DATA_BLOCK "DB3323"
TITLE =STAZIONE ++ZNE05
{ S7_language := '22(1) Portoghese (Brasile)  01.09.2016  10:42:20' }
VERSION : 0.1


  STRUCT
   CM_ID : STRING  [8 ] := '=DCK_2';	//COMPOSITE MACHINE
   STATION_ID : STRING  [8 ] := '++ZNE05';	//STATION - TRATTO - ZONE
   ELEMENT_ID : STRING  [8 ];	//ELEMENT
   DB_ID : INT  := 3;	//DB SIZE or TYPE
   PART_STYLE : STRING  [12 ];	//PART STYLE ON LAST STATION
   ACT_CYCLE_TIME : INT ;	//ACTUAL CYCLE TIME FOR THIS STYLE
   COUNT_GOOD : INT ;	//COUNTER GOOD PIECES
   COUNT_SCRAP : INT ;	//COUNTER SCRAP PIECES
   SPARE_00 : ARRAY  [0 .. 15 ] OF //SPARE INTEGER
   INT ;
   SPARE_01 : ARRAY  [0 .. 17 ] OF //SPARE INTEGER
   INT ;
   CODE_EVENT : ARRAY  [0 .. 7 ] OF INT ;
EVENTS : STRUCT
   E0000 : BOOL ;	//=DCK_2++ZNE05+PTZ01-SB_09;EMERGÊNCIA ATIVADA - NO PTZ01;2
   E0001 : BOOL ;	//=DCK_2++ZNE05+PTZ02-SB_09;EMERGÊNCIA ATIVADA - NO PTZ02;2
   E0002 : BOOL ;	//=DCK_2++ZNE05;EMERGÊNCIA NÃO RESTAURADA EM ++ZNE05;2
   E0003 : BOOL ;	//=DCK_2++ZNE05;ÁREAS DE AJUSTE DE EMERGÊNCIA ++ZNE05 (++ZNE04/6/7);2
   E0004 : BOOL ;	//=DCK_2++ZNE05+HCZ01-KM_06;FALHA DO CONTATO DO FREIO TR_01;1
   E0005 : BOOL ;	//=DCK_2++ZNE05+HCZ01-KM_08;FALHA NO CONTATO DO FREIO TR_02;1
   E0006 : BOOL ;	//=DCK_2++ZNE05+HCZ01-DMC01;ANOMALIA DO MÓDULO SEGURO ET200S-FDI-FDO;2
   E0007 : BOOL ;	//=DCK_2++ZNE05+HKM01-DMC01;ANOMALIA DO MÓDULO SEGURO ET200S-FDI;2
   E0008 : BOOL ;	//=DCK_2++ZNE05+PTZ01-DMC01;ANOMALIA DO MÓDULO SEGURO ET200S-FDI;2
   E0009 : BOOL ;	//=DCK_2++ZNE05+PTZ02-DMC01;ANOMALIA DO MÓDULO SEGURO ET200S-FDI;2
   E0010 : BOOL ;	//=DCK_2++ZNE05+HKM02-DMC01;ANOMALIA DO MÓDULO SEGURO ET200S-FDI;2
   E0011 : BOOL ;	//=DCK_2++ZNE05+HKM03-DMC01;ANOMALIA DO MÓDULO SEGURO ET200S-FDI;2
   E0012 : BOOL ;	//=DCK_2++ZNE05+HKM04-DMC01;ANOMALIA DO MÓDULO SEGURO ET200S-FDI;2
   E0013 : BOOL ;	//=DCK_2++ZNE05+HKM05-DMC01;ANOMALIA DO MÓDULO SEGURO ET200S-FDI;2
   E0014 : BOOL ;	//=DCK_2++ZNE05+HKM06-DMC01;ANOMALIA DO MÓDULO SEGURO ET200S-FDI;2
   E0015 : BOOL ;	//=DCK_2++ZNE05+HCZ01-DMC02;ANOMALIA DO MÓDULO SEGURO ET200S-FDO;2
   E0016 : BOOL ;	//=DCK_2++ZNE05+XGA01-SC_01;PORTÃO +XGA01 ++ZNE05 ABERTO;2
   E0017 : BOOL ;	//=DCK_2++ZNE05+XGA02-SC_01;PORTÃO +XGA02 ++ZNE05 ABERTO;2
   E0018 : BOOL ;	//=DCK_2++ZNE05+XGA01-SC_01;PORTÃO NÃO RESTAURADO PARA CICLO GM;2
   E0019 : BOOL ;	//=DCK_2++ZNE05+XGA02-SC_01;PORTÃO NÃO RESTAURADO PARA CICLO GM;2
   E0020 : BOOL ;	//=DCK_2++ZNE05+HCZ01-KA_17;FALHA DO RELÉ HABILITAÇÃO DO MOVIDRIVE PRX01-OP120;1
   E0021 : BOOL ;	//=DCK_2++ZNE05+HCZ01-KA_18;FALHA NO RELÉ DE HABILITAÇÃO DO MOVIDRIVE PRZ01-OP120;1
   E0022 : BOOL ;	//=DCK_2++ZNE05+HCZ01-KA_19;FALHA NO RELÉ DE HABILITAÇÃO DO MOVIDRIVE PRZ02-OP120;1
   E0023 : BOOL ;	//=DCK_2++ZNE05+HCZ01-KA_20;FALHA NO RELÉ DE HABILITAÇÃO DO MOVIDRIVE PRZ03-OP120;1
   E0024 : BOOL ;	//=DCK_2++ZNE05+HCZ01-KA_28;FALHA DO RELÉ HABILITAÇÃO DO MOVIDRIVE CRX03-OP130;1
   E0025 : BOOL ;	//=DCK_2++ZNE05+HCZ01-KA_29;FALHA DO RELÉ HABILITAÇÃO DO MOVIDRIVE CRX05-06-OP130;1
   E0026 : BOOL ;	//=DCK_2++ZNE05+HCZ01-KA_30;FALHA DO RELÉ HABILITAÇÃO DO MOVIDRIVE CRZ07-OP130;1
   E0027 : BOOL ;	//=DCK_2++ZNE05+HCZ01-KA_31;FALHA DO RELÉ HABILITAÇÃO DO MOVIDRIVE CRZ08-OP130;1
   E0028 : BOOL ;	//=DCK_2++ZNE05+HCZ01-KA_32;FALHA DO RELÉ HABILITAÇÃO DO MOVIDRIVE CRX04-OP130;1
   E0029 : BOOL ;	//=DCK_2++ZNE05+HCZ01-KA_33;FALHA DE RELÉ DE HABILITAÇÃO DO MOVIDRIVE CRY07-CRY08-OP130;1
   E0030 : BOOL ;	//=DCK_2++ZNE05+HCZ01-KA_34;FALHA DE RELÉ DE HABILITAÇÃO DO MOVID CRY09-OP130;1
   E0031 : BOOL ;	//=DCK_2++ZNE05+HCZ01-KA_35;FALHA DE RELÉ DE HABILITAÇÃO DO MOVID CRY10-OP130;1
   E0032 : BOOL ;	//=DCK_2++ZNE05+HCZ01-QF_73;ALIMENTAÇÃO DISJUNTOR TÉRMICO PARA CIRCUITOS AUXILIARES;1
   E0033 : BOOL ;	//=DCK_2++ZNE05+HCZ01-QF_75;FONTE DE ALIMENTAÇÃO MAGNETOTÉRMICA PARA CIRCUITOS DE SEGURANÇA;1
   E0034 : BOOL ;	//=DCK_2++ZNE05+HCZ01-QF_81;FONTE DE ALIMENTAÇÃO MAGNETOTÉRMICA +PTZ01;1
   E0035 : BOOL ;	//=DCK_2++ZNE05+HCZ01-QF_82;FONTE DE ALIMENTAÇÃO MAGNETOTÉRMICA +PTZ02;1
   E0036 : BOOL ;	//=DCK_2++ZNE05+HCZ01-QF_40;FONTE DE ALIMENTAÇÃO MAGNETOTÉRMICA. FREIOS 24VCC;1
   E0037 : BOOL ;	//=DCK_2++ZNE05+HCZ01-QF_41;FONTE DE ALIMENTAÇÃO MAGNETOTÉRMICA DE FREIO 24VDC;1
   E0038 : BOOL ;	//=DCK_2++ZNE05+HCZ01-QM_01;MOTOR DE ROLO DE MESA INVERSOR MAGNETOT +TR_01-OP120;1
   E0039 : BOOL ;	//=DCK_2++ZNE05+HCZ01-QF_02;MAGNETO. FREIO MOTOR DE ROLO DE MESA +TR_01-OP120;1
   E0040 : BOOL ;	//=DCK_2++ZNE05+HCZ01-QM_02;MOTOR DE ROLO DE MESA INVERSOR MAGNETOT +TR_02-OP130;1
   E0041 : BOOL ;	//=DCK_2++ZNE05+HCZ01-QF_03;MAGNETO. FREIO MOTOR DE ROLO DE MESA +TR_02 - OP130;1
   E0042 : BOOL ;	//=DCK_2++ZNE05+HCZ01-QF_83;MAGNETO. FORNECIMENTO DE GRUPOS DE VÁLVULAS;1
   E0043 : BOOL ;	//=DCK_2++ZNE05+HCZ01-QF_74;SINAIS DE COMANDOS DE SAÍDA DA FONTE DE ALIMENTAÇÃO MAGNETOT.;1
   E0044 : BOOL ;	//=DCK_2++ZNE05+HCZ01-QF_76;MAGNETO. FONTE DE ALIMENTAÇÃO PARA MÓDULOS DE E/S ET200S/PRO/ECO;1
   E0045 : BOOL ;	//=DCK_2++ZNE05+HCZ01-QF_82;CABEÇAS DE LEITURA DE FORNECIMENTO DE MAGNETO RF180C-OP130/135;1
   E0046 : BOOL ;	//=DCK_2++ZNE05+HCZ01-QF_31;MAGNETO. FONTE DE ALIMENTAÇÃO DO AR CONDICIONADO;1
   E0047 : BOOL ;	//=DCK_2++ZNE05+HCZ01-QF_85;MAGN. PODER SISTEMA ANTICOLISÃO +TR_01;1
   E0048 : BOOL ;	//=DCK_2++ZNE05+HCZ01-R_01;RESISTOR DE FREIO INVERSOR DE ROLO +TR_01-OP120;1
   E0049 : BOOL ;	//=DCK_2++ZNE05+TR_01-SQ_05;CONTROLE DE ROTAÇÃO TRASEIRA DAS CORREIAS DIREITAS - OP120;1
   E0050 : BOOL ;	//=DCK_2++ZNE05+TR_01-SQ_04;CONTROLE DE ROTAÇÃO TRASEIRA DAS CORREIAS ESQUERDAS - OP120;1
   E0051 : BOOL ;	//=DCK_2++ZNE05+HCZ01-U_02;ANOMALIA DO ROLO MOVIDRIVE +TR_02 - OP130;1
   E0052 : BOOL ;	//=DCK_2++ZNE05+HCZ01-U_01;ANOMALIA DO ROLO MOVIDRIVE +TR_01 - OP120;1
   E0053 : BOOL ;	//=DCK_2++ZNE05+TR_01-SQ_01;SEM PRESENÇA TRASEIRA NA MESA - OP120;1
   E0054 : BOOL ;	//=DCK_2++ZNE05+TR_01-SQ_03;MANCATA PRESENZA ANTERIORE SU TAVOLA - OP120 ;1
   E0055 : BOOL ;	//=DCK_2++ZNE05+HCZ01-R_02;RESISTIR. DE ROLOS DE MESA INVERSORA DE FREIO +TR_02-OP130;1
   E0056 : BOOL ;	//=DCK_2++ZNE05+TR_02-SQ_05;CONTROLE DE ROTAÇÃO TRASEIRA DAS CORREIAS DIREITAS - OP130;1
   E0057 : BOOL ;	//=DCK_2++ZNE05+TR_02-SQ_04;CONTROLE DE ROTAÇÃO TRASEIRA DAS CORREIAS ESQUERDAS - OP130;1
   E0058 : BOOL ;	//=DCK_2++ZNE05+TR_02-SQ_06/7;INEFEITO. CENTRO DE SKID DE PARADA ALTA/BAIXA NO OP130;1
   E0059 : BOOL ;	//=DCK_2++ZNE05+PCV02-SP_01;CONTROLE DE PRESSÃO DE AR ??- OP130;1
   E0060 : BOOL ;	//=DCK_2++ZNE05+PCV02-SP_02;CIRCUITO DE LIBERAÇÃO MANUAL DO ATUADOR OP130 DE CONTROLE DE PRESSÃO DE AR;1
   E0061 : BOOL ;	//=DCK_2++ZNE05+SID01-D_01;ANOMALIA DA CABEÇA DE LEITURA EM +TR_02 OP130;1
   E0062 : BOOL ;	//=DCK_2++ZNE05+SID01-D_01;LEITURA DE DADOS INCORRETOS NA CABEÇA DE LEITURA OP130;1
   E0063 : BOOL ;	//=DCK_2++ZNE05+TR_02-SQ_01;FALHA NA LER DA LENTAÇÃO TRASEIRA - OP130;1
   E0064 : BOOL ;	//=DCK_2++ZNE05+TR_01;TEMPO LIMITE DE TRANSFERÊNCIA +TR_01->+TR_02 ++ZNE05;1
   E0065 : BOOL ;	//=DCK_2++ZNE05+TR_02;TEMPO LIMITE DE TRANSFERÊNCIA +TR_02->+TR_01 ++ZNE06;1
   E0066 : BOOL ;	//=DCK_2++ZNE05+TR_02-SQ_06/7;TIME OUT SKID CENTER ALTO EM +TR_02;1
   E0067 : BOOL ;	//=DCK_2++ZNE05+TR_02-SQ_06/7;TIME OUT SKID CENTER BAIXO EM +TR_02;1
   E0068 : BOOL ;	//=DCK_2++ZNE05+SID01-D_01;OP130 TEMPO LIMITE DE LEITURA/ESCRITA DA CABEÇA DE LEITURA;1
   E0069 : BOOL ;	//=DCK_2++ZNE05+SID01-D_01;OP120 TEMPO LIMITE DE LEITURA/ESCRITA DA CABEÇA DE LEITURA;1
   E0070 : BOOL ;	//=DCK_2++ZNE05+PTZ01-SA_03;PEDIDO DE ABERTURA DE PORTÃO +XGA01 PARA CICLO PM;13
   E0071 : BOOL ;	//=DCK_2++ZNE05+PTZ02-SA_03;PEDIDO DE ABERTURA DE PORTÃO +XGA02 PARA CICLO PM;13
   E0072 : BOOL ;	//=DCK_2++ZNE05+TR_01-SQ_06/7;INEFEITO. CENTRO DE SKID DE PARADA ALTA/BAIXA NO OP120;1
   E0073 : BOOL ;	//=DCK_2++ZNE05+TR_01-SQ_06/7;TIME OUT SKID CENTER ALTO EM +TR_01;1
   E0074 : BOOL ;	//=DCK_2++ZNE05+TR_01-SQ_06/7;TIME OUT SKID CENTER BAIXO EM +TR_01;1
   E0075 : BOOL ;	//=DCK_2++ZNE05+PRX02-QM_20;MOTOR PORTAL INVERSOR MAGNÉTICO TÉRMICO +PRX02 OP120;1
   E0076 : BOOL ;	//=DCK_2++ZNE05+PRX02-QF_60;ÍMÃ TÉRMICO DE FREIO MOTOR PORTAL +PRX02 OP120;1
   E0077 : BOOL ;	//=DCK_2++ZNE05+SWK_OP120;TEMPO LIMITE DO CICLO DA CHAVE DE FENDA OP120;1
   E0078 : BOOL ;	//=DCK_2++ZNE05+SWK_OP130;TEMPO LIMITE DO CICLO DA CHAVE DE FENDA OP130;1
   E0079 : BOOL ;	//=DCK_2++ZNE05+HCZ01-KA_36;FALHA NO RELÉ DE HABILITAÇÃO DO MOVIDRIVE CRY11-OP130;1
   E0080 : BOOL ;	//=DCK_2++ZNE05+PTZ02;PARAFUSOS DESATIVADOS DO PAINEL +PTZ02;55
   E0081 : BOOL ;	//=DCK_2++ZNE05+HCZ01-KA_37;FALHA NO RELÉ DE HABILITAÇÃO DO MOVIDRIVE CRY12-OP130;1
   E0082 : BOOL ;	//=DCK_2++ZNE05+PTZ01-SA_03;PEDIDO DE ABERTURA DE PORTÃO +XGA01 PARA CICLO AM;14
   E0083 : BOOL ;	//=DCK_2++ZNE05+PTZ02-SA_03;PEDIDO DE ABERTURA DE PORTÃO +XGA02 PARA CICLO AM;14
   E0084 : BOOL ;	//=DCK_2++ZNE05+TR_01;FALHA AO DESCARREGAR TABELA +TR_01 OP120;9
   E0085 : BOOL ;	//=DCK_2++ZNE05+TR_02;FALHA AO DESCARREGAR TABELA +TR_02 OP130;9
   E0086 : BOOL ;	//=DCK_2++ZNE05;CICLO NÃO INICIADO ZONA ++ZNE05;15
   E0087 : BOOL ;	//=DCK_2++ZNE05;CONDIÇÕES DE INICIALIZAÇÃO DO SISTEMA FALTA PAINEL GERAL ++PRINCIPAL+HGD01;15
   E0088 : BOOL ;	//=DCK_2++ZNE05;PAINEL GERAL DE EMERGÊNCIA ++PRINCIPAL+HGD01;2
   E0089 : BOOL ;	//=DCK_2++ZNE05;CICLO NÃO INICIADO NO CONTROLE PRINCIPAL ++PRINCIPAL+HGD01;15
   E0090 : BOOL ;	//=DCK_2++ZNE05;CICLO NÃO INICIADO CHAVE DE FENDA ÁREA INFERIOR OP130++ZNE05;15
   E0091 : BOOL ;	//=DCK_2++ZNE05;CICLO NÃO INICIADO ÁREA INFERIOR DA MOLA OP120 ++ZNE05;15
   E0092 : BOOL ;	//=DCK_2++ZNE05;PARADA DE CICLO DO CONTROLE PRINCIPAL ++PRINCIPAL+HGD01;17
   E0093 : BOOL ;	//=DCK_2++ZNE05;PARADA DO CICLO DA ZONA ++ZNE05;17
   E0094 : BOOL ;	//=DCK_2++ZNE05;PARADA DE CICLO ÁREA INFERIOR OP130 ++ZNE05 CHAVES DE FENDA;17
   E0095 : BOOL ;	//=DCK_2++ZNE05;PARADA DE CICLO ÁREA INFERIOR PLANTA DE MOLA OP120 ++ZNE05;17
   E0096 : BOOL ;	//=DCK_2++ZNE05+TR_02-SQ_03;FALHA NA LEITURA DA LENTAÇÃO FRONTAL - OP130;1
   E0097 : BOOL ;	//=DCK_2++ZNE05+SID01-D_01;ANOMALIA DA CABEÇA DE LEITURA EM +TR_01 OP120;1
   E0098 : BOOL ;	//=DCK_2++ZNE05+SID01-D_01;LEITURA DE DADOS INCORRETOS NA CABEÇA DE LEITURA OP120;1
   E0099 : BOOL ;	//=DCK_2++ZNE05+TR_01-B_01;FALHA DE FOTOCÉLULA DE DADOS AVANÇADOS +EPT01 OP120;1
   E0100 : BOOL ;	//=DCK_2++ZNE05+TR_01;FALHA NO CARREGAMENTO DA TABELA +TR_01 OP120;6
   E0101 : BOOL ;	//=DCK_2++ZNE05+TR_02;FALHA NO CARREGAMENTO DA TABELA +TR_02 OP130;6
   E0102 : BOOL ;	//=DCK_2++ZNE05+TR_01;TABELA +TR_01 OP120 BLOQUEADA PELA TABELA +TR_02 OP130;58
   E0103 : BOOL ;	//=DCK_2++ZNE05+TR_02;TABELA +TR_02 OP130 BLOQUEADA PELA TABELA +TR_01 OP135;58
   E0104 : BOOL ;	//=DCK_2++ZNE05+TR_01-SE_02;LEITOR TRASEIRO -SKID DE CÓDIGO DE BARRAS DESCONTINUADO OP120;1
   E0105 : BOOL ;	//=DCK_2++ZNE05+TR_01-SE_03;LEITOR FRONTAL -SKID DE CÓDIGO DE BARRAS DESCONTINUADO OP120;1
   E0106 : BOOL ;	//=DCK_2++ZNE05+TR_01-SE_02;LEITOR TRASEIRO - PRESENÇA SUJA OP120;58
   E0107 : BOOL ;	//=DCK_2++ZNE05+TR_01-SE_03;LEITOR FRONTAL - PRESENÇA SUJA OP120;58
   E0108 : BOOL ;	//=DCK_2++ZNE05+TR_01-SE_02;LEITOR TRASEIRO EM ERRO OP120;1
   E0109 : BOOL ;	//=DCK_2++ZNE05+TR_01-SE_03;LEITOR FRONTAL EM ERRO OP120;1
   E0110 : BOOL ;	//=DCK_2++ZNE05+TR_01-SE_02;LEITOR TRASEIRO - COTA DE FAIXA NÃO OK OP120;1
   E0111 : BOOL ;	//=DCK_2++ZNE05+TR_01-SE_03;LEITOR FRONTAL - COTA DE FAIXA NÃO OK OP120;1
   E0112 : BOOL ;	//=DCK_2++ZNE05+HCZ01-QF_86;MAGN. FONTE DE ENERGIA SISTEMA ANTICOLISÃO +TR_02;58
   E0113 : BOOL ;	//=DCK_2++ZNE05+HCZ01-DMC01;GABINETE ELÉTRICO NODE 6 PROFINET ET200S;1
   E0114 : BOOL ;	//=DCK_2++ZNE05+PTZ01-DMC01;PAINEL BOTÃO NODE 14 PROFINET ET200S;1
   E0115 : BOOL ;	//=DCK_2++ZNE05+PTZ02-DMC01;PAINEL BOTÃO NODE 15 PROFINET ET200S;1
   E0116 : BOOL ;	//=DCK_2++ZNE05+TR_01-DMC01;NÓ 62 PROFINET ET200ECO +TR_01;1
   E0117 : BOOL ;	//=DCK_2++ZNE05+TR_02-DMC01;NÓ 63 PROFINET ET200ECO +TR_02;1
   E0118 : BOOL ;	//=DCK_2++ZNE05+HCZ01-DSW01;ARMÁRIO ELÉTRICO NODE 240 PROFINET SCALANCE;58
   E0119 : BOOL ;	//=DCK_2++ZNE05+HCZ01-DSW02;GABINETE ELÉTRICO NODE 246 PROFINET SCALANCE;58
   E0120 : BOOL ;	//=DCK_2++ZNE05+PCV01-DMC01;PACOTE DE VÁLVULAS NODE 229 PROFINET FESTO OP120;58
   E0121 : BOOL ;	//=DCK_2++ZNE05+PCV02-DMC01;PACOTE DE VÁLVULAS NODE 233 PROFINET FESTO OP130;58
   E0122 : BOOL ;	//=DCK_2++ZNE05+SID02-D_01;NÓ 137 LEITOR PROFINET RF180R MOBY OP130;58
   E0123 : BOOL ;	//=DCK_2++ZNE05+SID01-D_01;LEITOR PROFINET NÓ 132 RF180R MOBY OP120;58
   E0124 : BOOL ;	//=DCK_2++ZNE05+DPM01-DMC01;NÓ 93 PROFINET ET200PRO OP120;1
   E0125 : BOOL ;	//=DCK_2++ZNE05+HCZ01-KA 21;FALHA DO RELÉ HABILITAÇÃO DO MOVIDRIVE PRX02-OP130;1
   E0126 : BOOL ;	//=DCK_2++ZNE05+HCZ01-KA_41;FALHA NO RELÉ DE HABILITAÇÃO DO MOVIDRIVE PRY01-OP130;1
   E0127 : BOOL ;	//=DCK_2++ZNE05+HCZ01-KA_42;FALHA NO RELÉ DE HABILITAÇÃO DO MOVIDRIVE PRY02-OP130;1
   E0128 : BOOL ;	//=DCK_2++ZNE05;OP120->OP130 SISTEMA ANTICOLISÃO DISPARADO;1
   E0129 : BOOL ;
   E0130 : BOOL ;
   E0131 : BOOL ;	//=DCK_2++ZNE05+TR_01-SE_02;LEITOR TRASEIRO - ANOMALIA DE ATUALIZAÇÃO DE COTA OP120;1
   E0132 : BOOL ;	//=DCK_2++ZNE05+TR_01-SE_03;LEITOR FRONTAL - ANOMALIA DE ATUALIZAÇÃO DE COTA OP120;1
   E0133 : BOOL ;	//=DCK_2++ZNE05+TR_02-SE_02;LEITOR TRASEIRO -SKID DE CÓDIGO DE BARRAS DESCONTINUADO OP130;1
   E0134 : BOOL ;	//=DCK_2++ZNE05+TR_02-SE_03;LEITOR FRONTAL -SKID DE CÓDIGO DE BARRAS DESCONTINUADO OP130;1
   E0135 : BOOL ;	//=DCK_2++ZNE05+TR_02-SE_02;LEITOR TRASEIRO - PRESENÇA SUJA OP130;58
   E0136 : BOOL ;	//=DCK_2++ZNE05+TR_02-SE_03;LEITOR FRONTAL - PRESENÇA SUJA OP130;58
   E0137 : BOOL ;	//=DCK_2++ZNE05+TR_02-SE_02;LEITOR TRASEIRO EM ERRO OP130;1
   E0138 : BOOL ;	//=DCK_2++ZNE05+TR_02-SE_03;LEITOR FRONTAL EM ERRO OP130;1
   E0139 : BOOL ;	//=DCK_2++ZNE05+TR_02-SE_02;LEITOR TRASEIRO - FAIXA DE ALTURA NÃO OK OP130;1
   E0140 : BOOL ;	//=DCK_2++ZNE05+TR_02-SE_03;LEITOR FRONTAL - FAIXA DE ALTURA NÃO OK OP130;1
   E0141 : BOOL ;	//=DCK_2++ZNE05;OP130->OP135 SISTEMA ANTICOLISÃO DISPARADO;1
   E0142 : BOOL ;
   E0143 : BOOL ;
   E0144 : BOOL ;	//=DCK_2++ZNE05+TR_02-SE_02;LEITOR TRASEIRO - ANOMALIA DE ATUALIZAÇÃO DE COTA OP130;1
   E0145 : BOOL ;	//=DCK_2++ZNE05+TR_02-SE_03;LEITOR FRONTAL - ANOMALIA DE ATUALIZAÇÃO DE COTA OP130;1
   E0146 : BOOL ;	//=DCK_2++ZNE05;LEITOR ANTICOLISÃO ++ZNE05 DESATIVADO;54
   E0147 : BOOL ;	//=DCK_2++ZNE05+TR_01-SQ_02;FALHA NA LER LENTAÇÃO EM +TR_01 OP120;1
   E0148 : BOOL ;	//=DCK_2++ZNE05+TR_02-SQ_02;FALHA NA LER LENTAÇÃO EM +TR_02 OP130;1
   E0149 : BOOL ;
   E0150 : BOOL ;
   E0151 : BOOL ;
   E0152 : BOOL ;	//=DCK_2++ZNE05+HCZ01-KA_01/02;SÉRIE DE FEEDBACK DE EMERGÊNCIA "E82.6" (CAT.1)++ZNE05;2
   E0153 : BOOL ;	//=DCK_2++ZNE05+HCZ01-KA_03/04;SÉRIE DE FEEDBACK DE EMERGÊNCIA "E82.7" (CAT.0)++ZNE05;2
   E0154 : BOOL ;	//=DCK_2++ZNE05+HCZ01-KA_05;SÉRIE FEEDBACK HABILITA MOVIDRIVE +TR_01 OP120;2
   E0155 : BOOL ;	//=DCK_2++ZNE05+HCZ01-KA_06;SÉRIE FEEDBACK HABILITA MOVIDRIVE +TR_02 OP130;2
   E0156 : BOOL ;	//=DCK_2++ZNE05+HCZ01-KA_07;SÉRIE FEEDBACK HABILITA MOVIDRIVE +CRX01 OP130;2
   E0157 : BOOL ;	//=DCK_2++ZNE05+HCZ01-KA_08;FEEDBACK ATIVAR MOVIDRIVE +CRY01/+CRY02 OP130;2
   E0158 : BOOL ;	//=DCK_2++ZNE05+HCZ01-KA_09;SÉRIE FEEDBACK HABILITA MOVIDRIVE +CRZ01 OP130;2
   E0159 : BOOL ;	//=DCK_2++ZNE05+HCZ01-KA_10;SÉRIE FEEDBACK HABILITA MOVIDRIVE +CRZ02 OP130;2
   E0160 : BOOL ;	//=DCK_2++ZNE05+HCZ01-KA_11;SÉRIE FEEDBACK HABILITA MOVIDRIVE +CRX02 OP130;2
   E0161 : BOOL ;	//=DCK_2++ZNE05+HCZ01-KA_12;FEEDBACK ATIVAR MOVIDRIVE +CRY03/+CRY04 OP130;2
   E0162 : BOOL ;	//=DCK_2++ZNE05+HCZ01-KA_13;SÉRIE FEEDBACK HABILITA MOVIDRIVE +CRZ03 OP130;2
   E0163 : BOOL ;	//=DCK_2++ZNE05+HCZ01-KA_14;SÉRIE FEEDBACK HABILITA MOVIDRIVE +CRZ04 OP130;2
   E0164 : BOOL ;	//=DCK_2++ZNE05+HCZ01-KA_17;SÉRIE FEEDBACK HABILITA MOVIDRIVE +PRX01 OP120;2
   E0165 : BOOL ;	//=DCK_2++ZNE05+HCZ01-KA_18;SÉRIE DE FEEDBACK ATIVAR..MOVIDRIVE +PRZ01 OP120;2
   E0166 : BOOL ;	//=DCK_2++ZNE05+HCZ01-KA_19;SÉRIE FEEDBACK HABILITA MOVIDRIVE +PRZ02 OP120;2
   E0167 : BOOL ;	//=DCK_2++ZNE05+HCZ01-KA_20;SÉRIE FEEDBACK HABILITA MOVIDRIVE +PRZ03 OP120;2
   E0168 : BOOL ;	//=DCK_2++ZNE05+HCZ01-KA_21;SÉRIE FEEDBACK HABILITA MOVIDRIVE +PRX02 OP120;2
   E0169 : BOOL ;
   E0170 : BOOL ;
   E0171 : BOOL ;
   E0172 : BOOL ;
   E0173 : BOOL ;
   E0174 : BOOL ;
   E0175 : BOOL ;
   E0176 : BOOL ;	//=DCK_2++ZNE05+HCZ01-U_01;AVISO ROLOS MOVIDRIVE +TR_01 - OP120;58
   E0177 : BOOL ;	//=DCK_2++ZNE05+HCZ01-U_02;AVISO ROLOS MOVIDRIVE +TR_02 - OP130;58
   E0178 : BOOL ;
   E0179 : BOOL ;
   E0180 : BOOL ;
   E0181 : BOOL ;
   E0182 : BOOL ;
   E0183 : BOOL ;
   E0184 : BOOL ;
   E0185 : BOOL ;
   E0186 : BOOL ;
   E0187 : BOOL ;
   E0188 : BOOL ;
   E0189 : BOOL ;
   E0190 : BOOL ;
   E0191 : BOOL ;
   E0192 : BOOL ;	//=DCK_2++ZNE05+PCV01-SP_01;OP120 INTERRUPTOR DE PRESSÃO DE CONTROLE DE PRESSÃO DE AR;1
   E0193 : BOOL ;	//=DCK_2++ZNE05+PCV01-SP_02;CIRCUITO DE LIBERAÇÃO MANUAL DO ATUADOR OP120 DE CONTROLE DE PRESSÃO DE AR;1
   E0194 : BOOL ;	//=DCK_2++ZNE05+DPM01-SQ_01/02;MAU FUNCIONAMENTO DO INTERRUPTOR DE LIMITE DE POSIÇÃO DO CILINDRO C01 OP120;1
   E0195 : BOOL ;	//=DCK_2++ZNE05+DPM01-SQ_03/04;MAU FUNCIONAMENTO DO INTERRUPTOR DE LIMITE DE POSIÇÃO DO CILINDRO C02 OP120;1
   E0196 : BOOL ;	//=DCK_2++ZNE05+DPM01-SQ_05/06;MAU FUNCIONAMENTO DO INTERRUPTOR DE LIMITE DE POSIÇÃO DO CILINDRO C05 OP120;1
   E0197 : BOOL ;	//=DCK_2++ZNE05+DPM01-SQ_07/08;MAU FUNCIONAMENTO DO INTERRUPTOR DE LIMITE DE POSIÇÃO DO CILINDRO C06 OP120;1
   E0198 : BOOL ;	//=DCK_2++ZNE05+DPM01-SQ_09/10;MAU FUNCIONAMENTO DO INTERRUPTOR DE LIMITE DE POSIÇÃO DO CILINDRO C09 OP120;1
   E0199 : BOOL ;	//=DCK_2++ZNE05+DPM01-SQ_11/12;MAU FUNCIONAMENTO DO INTERRUPTOR DE LIMITE DE POSIÇÃO DO CILINDRO C10 OP120;1
   E0200 : BOOL ;	//=DCK_2++ZNE05+DPM01-SQ_13/14;MAU FUNCIONAMENTO DO INTERRUPTOR DE LIMITE DE POSIÇÃO DO CILINDRO C11 OP120;1
   E0201 : BOOL ;	//=DCK_2++ZNE05+DPM01-SQ_15/16;MAU FUNCIONAMENTO DO INTERRUPTOR DE LIMITE DE POSIÇÃO DO CILINDRO C12 OP120;1
   E0202 : BOOL ;	//=DCK_2++ZNE05+DPM01-SQ_17/18;MAU FUNCIONAMENTO DO INTERRUPTOR DE LIMITE DE POSIÇÃO DO CILINDRO C13 OP120;1
   E0203 : BOOL ;	//=DCK_2++ZNE05+DPM01;TIME OUT POSICIONAMENTO DO CILINDRO DA PLANTA C01/2 OP120;1
   E0204 : BOOL ;	//=DCK_2++ZNE05+DPM01;TIME OUT POSICIONAMENTO DO CILINDRO DA PLANTA C05/6 OP120;1
   E0205 : BOOL ;	//=DCK_2++ZNE05+DPM01;TIME OUT POSICIONAMENTO DO CILINDRO DA PLANTA C09/10 OP120;1
   E0206 : BOOL ;	//=DCK_2++ZNE05+DPM01;TIME OUT POSICIONAMENTO DO CILINDRO DA PLANTA C11/12/13 OP120;1
   E0207 : BOOL ;
   E0208 : BOOL ;	//=DCK_2++ZNE05+PRZ01-SQ_03;HASTE DE CHAVE DE FENDA DE VIAGEM EXTRA NO SLIDE +PRZ01 OP120;1
   E0209 : BOOL ;	//=DCK_2++ZNE05+PRZ02-SQ_03;CHAVE DE FENDA EXTRA VIAGEM HASTE 1 SLIDE +PRZ02 OP120;1
   E0210 : BOOL ;	//=DCK_2++ZNE05+PRZ02-SQ_04;VIAGEM EXTRA PARA HASTE CHAVE DE FENDA 2 SLIDE +PRZ02 OP120;1
   E0211 : BOOL ;	//=DCK_2++ZNE05+PRZ02-SQ_05;CHAVE DE FENDA EXTRA VIAGEM HASTE 3 DESLIZAMENTO +PRZ02 OP120;1
   E0212 : BOOL ;	//=DCK_2++ZNE05+PRZ02-SQ_06;CHAVE DE FENDA EXTRA VIAGEM HASTE 4 DESLIZAMENTO +PRZ02 OP120;1
   E0213 : BOOL ;	//=DCK_2++ZNE05+PRZ03-SQ_03;CHAVE DE FENDA EXTRA VIAGEM HASTE 1 SLIDE +PRZ03 OP120;1
   E0214 : BOOL ;	//=DCK_2++ZNE05+PRZ03-SQ_04;VIAGEM EXTRA PARA HASTE CHAVE DE FENDA 2 SLIDE +PRZ03 OP120;1
   E0215 : BOOL ;	//=DCK_2++ZNE05+PRZ03-SQ_05;CHAVE DE FENDA EXTRA VIAGEM HASTE 3 DESLIZAMENTO +PRZ03 OP120;1
   E0216 : BOOL ;	//=DCK_2++ZNE05+PRZ03-SQ_06;CHAVE DE FENDA EXTRA VIAGEM HASTE 4 SLIDE +PRZ03 OP120;1
   E0217 : BOOL ;	//=DCK_2++ZNE05+PRX01-SQ_01;PORTAL AVANÇAR VIAGEM EXTRA +PRX02 OP120;1
   E0218 : BOOL ;	//=DCK_2++ZNE05+PRX01-SQ_02;PORTAL BACKWARD VIAGEM EXTRA +PRX02 OP120;1
   E0219 : BOOL ;
   E0220 : BOOL ;
   E0221 : BOOL ;
   E0222 : BOOL ;
   E0223 : BOOL ;
   E0224 : BOOL ;
   E0225 : BOOL ;
   E0226 : BOOL ;
   E0227 : BOOL ;
   E0228 : BOOL ;
   E0229 : BOOL ;
   E0230 : BOOL ;
   E0231 : BOOL ;
   E0232 : BOOL ;
   E0233 : BOOL ;
   E0234 : BOOL ;
   E0235 : BOOL ;
   E0236 : BOOL ;
   E0237 : BOOL ;
   E0238 : BOOL ;
   E0239 : BOOL ;
   E0240 : BOOL ;	//=DCK_2++ZNE05;PRODUÇÃO++ZNE05;19
   E0241 : BOOL ;	//=DCK_2++ZNE05+PTZ01-SA_01;ZONA DE CICLO MANUAL ++ZNE05 ON +PTZ01;16
   E0242 : BOOL ;	//=DCK_2++ZNE05+PTZ02-SA_01;ZONA DE CICLO MANUAL ++ZNE05 ON +PTZ02;16
   E0243 : BOOL ;	//=DCK_2++ZNE05+PTZ01;PEDIDO DE ABERTURA DE PORTÃO +XGA01 PARA CICLO GM;58
   E0244 : BOOL ;	//=DCK_2++ZNE05+PTZ02;PEDIDO DE ABERTURA DE PORTÃO +XGA02 PARA CICLO GM;58
   E0245 : BOOL ;	//=DCK_2++ZNE05+XGA01-SC_01;PORTÃO NÃO RESTAURADO PARA CICLO AM;13
   E0246 : BOOL ;	//=DCK_2++ZNE05+XGA01-SC_01;PORTÃO NÃO RESTAURADO PARA CICLO PM;14
   E0247 : BOOL ;	//=DCK_2++ZNE05+XGA02-SC_01;PORTÃO NÃO RESTAURADO PARA CICLO AM;13
   E0248 : BOOL ;	//=DCK_2++ZNE05+XGA02-SC_01;PORTÃO NÃO RESTAURADO PARA CICLO PM;14
   E0249 : BOOL ;
   E0250 : BOOL ;
   E0251 : BOOL ;
   E0252 : BOOL ;
   E0253 : BOOL ;
   E0254 : BOOL ;
   E0255 : BOOL ;
   E0256 : BOOL ;	//=DCK_2++ZNE05+HCZ01-QF_77;MAGNETO. PODER INVERSOR OP120-130;1
   E0257 : BOOL ;	//=DCK_2++ZNE05+HCZ01-QF_78;MAGNETO. FONTE DE ALIMENTAÇÃO INVERSOR PARA TRANSPORTE +CRX01;1
   E0258 : BOOL ;	//=DCK_2++ZNE05+HCZ01-QF_79;MAGNETO. FONTE DE ALIMENTAÇÃO INVERSOR PARA TRANSPORTE +CRX02;1
   E0259 : BOOL ;
   E0260 : BOOL ;	//=DCK_2++ZNE05+HCZ01-QM_03;MAGNETO. INVERSOR DE TRADUÇÃO DE CARRO +CRX01 -OP130;1
   E0261 : BOOL ;	//=DCK_2++ZNE05+HCZ01-QF_42;MAGNETO. FREIO MOTOR DE TRADUÇÃO +CRX01 -OP130;1
   E0262 : BOOL ;	//=DCK_2++ZNE05+HCZ01-QM_04;MAGN. DESLIZAR INVERSÃO. +CRY01 PARAFUSO ESQUERDO. +CRX01-OP130;1
   E0263 : BOOL ;	//=DCK_2++ZNE05+HCZ01-QF_43;MAGN.BRAKE SLIDE +CRY01 PARAFUSO ESQUERDO. +CRX01-OP130;1
   E0264 : BOOL ;	//=DCK_2++ZNE05+HCZ01-QM_06;MAGNET.REVERSE SLIDE +CRZ01 PARAFUSANDO À ESQUERDA. +CRX01-OP130;1
   E0265 : BOOL ;	//=DCK_2++ZNE05+HCZ01-QF_45;MAGN.FREIO MOSLITTA +CRZ01 PARAFUSO ESQUERDO.PARA CIMA +CRX01-OP130;1
   E0266 : BOOL ;	//=DCK_2++ZNE05+HCZ01-QM_05;MAGN. INVER. SLIDE +CRY02 PARAFUSAMENTO DIREITO. +CRX01 OP130;1
   E0267 : BOOL ;	//=DCK_2++ZNE05+HCZ01-QF_44;MAGN.BRAKE MOT.SLIDE +CRY02 PARAFUSO DIREITO. +CRX01 OP130;1
   E0268 : BOOL ;	//=DCK_2++ZNE05+HCZ01-QM_07;MAGN.INVER. DESLIZAMENTO + PARAFUSO CRZ02. DX. +CRX01 -OP130;1
   E0269 : BOOL ;	//=DCK_2++ZNE05+HCZ01-QF_46;DESLIZAMENTO DO MOTOR DE FREIO MAGN. +CRZ02 PARAFUSO DIREITO.+CRX01 OP130;1
   E0270 : BOOL ;	//=DCK_2++ZNE05+HCZ01-QM_08;MAGNETO. INVERSOR DE TRADUÇÃO DE CARRO +CRX02 - OP130;1
   E0271 : BOOL ;	//=DCK_2++ZNE05+HCZ01-QF_47;MAGNETO. FREIO DO MOTOR TRADUÇÃO DE CARRIAGE +CRX02-OP130;1
   E0272 : BOOL ;	//=DCK_2++ZNE05+HCZ01-U_03;CARRO MOVIDRIVE +CRX01 NÃO RESET - OP130;58
   E0273 : BOOL ;	//=DCK_2++ZNE05+HCZ01-U_03;TRANSPORTE DE ANOMALIA MOVIDRIVE +CRX01 - OP130;1
   E0274 : BOOL ;	//=DCK_2++ZNE05+CRX01-SQ_05;ANTICOLISÃO ENTRE +CRX01 E +CRX03 - CARROS OP130;1
   E0275 : BOOL ;	//=DCK_2++ZNE05+HCZ01-U_04;MOVIDRIVE SLIDE +CRY01 NÃO RESET - OP130;58
   E0276 : BOOL ;	//=DCK_2++ZNE05+HCZ01-U_04;ANOMALIA DO SLIDE MOVIDRIVE +CRY01 - OP130;1
   E0277 : BOOL ;	//=DCK_2++ZNE05+CRY01-SQ_01;CODIFICADOR EXTRA VIAGEM REVERSE/ZERO SLIDE - OP130;1
   E0278 : BOOL ;	//=DCK_2++ZNE05+CRY01-SQ_02;ANTICOLISÃO ENTRE SLIDES +CRY01 E +CRY02 - OP130;1
   E0279 : BOOL ;	//=DCK_2++ZNE05+HCZ01-U_06;ANOMALIA DO SLIDE MOVIDRIVE +CRZ01 - OP130;1
   E0280 : BOOL ;	//=DCK_2++ZNE05+CRZ01-SQ_01;EXTRACORSA ALTO SLITTA +CRZ01 - OP130 ;1
   E0281 : BOOL ;	//=DCK_2++ZNE05+CRZ01-SQ_02;CODIFICADOR DE SLIDE DE VIAGEM EXTRA BAIXO/ZERO - OP130;1
   E0282 : BOOL ;	//=DCK_2++ZNE05+CRZ01-SQ_03;CHAVE DE FENDA EXTRA DE VIAGEM NO SLIDE +CRZ01 - OP130;1
   E0283 : BOOL ;	//=DCK_2++ZNE05+HCZ01-U_05;MOVIDRIVE SLIDE +CRY02 NÃO RESET - OP130;58
   E0284 : BOOL ;	//=DCK_2++ZNE05+HCZ01-U_05;ANOMALIA DO SLIDE MOVIDRIVE +CRY02 - OP130;1
   E0285 : BOOL ;	//=DCK_2++ZNE05+CRY02-SQ_01;CODIFICADOR EXTRA VIAGEM REVERSE/ZERO SLIDE - OP130;1
   E0286 : BOOL ;	//=DCK_2++ZNE05+CRY01-SQ_02;ANTICOLISÃO ENTRE SLIDES +CRY01 E +CRY02 - OP130;1
   E0287 : BOOL ;	//=DCK_2++ZNE05+HCZ01-U_07;ANOMALIA DO SLIDE MOVIDRIVE +CRZ02 - OP130;1
   E0288 : BOOL ;	//=DCK_2++ZNE05+CRX01;TIME-OUT POSICIONAMENTO DO CARRO +CRX01 OP130;1
   E0289 : BOOL ;	//=DCK_2++ZNE05+CRY01;POSICIONAMENTO AUTOMÁTICO DO SLIDE TIME-OUT +CRY01 OP130;1
   E0290 : BOOL ;	//=DCK_2++ZNE05+CRZ01;POSICIONAMENTO AUTOMÁTICO DO SLIDE TIME-OUT +CRZ01 OP130;1
   E0291 : BOOL ;	//=DCK_2++ZNE05+CRY02;POSICIONAMENTO AUTOMÁTICO DO SLIDE TIME-OUT +CRY02 OP130;1
   E0292 : BOOL ;	//=DCK_2++ZNE05+CRZ02;POSICIONAMENTO AUTOMÁTICO DO SLIDE TIME-OUT +CRZ02 OP130;1
   E0293 : BOOL ;	//=DCK_2++ZNE05+CRX02;TIME-OUT POSICIONAMENTO AUTOMÁTICO DO CARRO +CRX02 OP130;1
   E0294 : BOOL ;	//=DCK_2++ZNE05+CRY03;POSICIONAMENTO AUTOMÁTICO DO SLIDE TIME-OUT +CRY03 OP130;1
   E0295 : BOOL ;	//=DCK_2++ZNE05+CRZ03;TEMPO LIMITE DE POSICIONAMENTO AUTOMÁTICO DO SLIDE +CRZ03 OP130;1
   E0296 : BOOL ;	//=DCK_2++ZNE05+CRY04;POSICIONAMENTO AUTOMÁTICO DO SLIDE TIME-OUT +CRY04 OP130;1
   E0297 : BOOL ;	//=DCK_2++ZNE05+CRZ04;TEMPO LIMITE DE POSICIONAMENTO AUTOMÁTICO DO SLIDE +CRZ04 OP130;1
   E0298 : BOOL ;	//=DCK_2++ZNE05+PRX01;TEMPO LIMITE DE POSICIONAMENTO AUTOMÁTICO DO PORTAL +PRX01-OP120;1
   E0299 : BOOL ;	//=DCK_2++ZNE05+PRZ01;POSICIONAMENTO AUTOMÁTICO DO SLIDE TIME-OUT +PRZ01 OP120;1
   E0300 : BOOL ;	//=DCK_2++ZNE05+CRZ05;POSICIONAMENTO AUTOMÁTICO DO SLIDE TIME-OUT +CRZ05 OP130;1
   E0301 : BOOL ;	//=DCK_2++ZNE05+PRZ02;TEMPO LIMITE DE POSICIONAMENTO AUTOMÁTICO DO SLIDE +PRZ02 OP120;1
   E0302 : BOOL ;	//=DCK_2++ZNE05+CRZ06;TEMPO LIMITE DE POSICIONAMENTO AUTOMÁTICO DO SLIDE +CRZ06 OP130;1
   E0303 : BOOL ;	//=DCK_2++ZNE05+PRZ03;TEMPO LIMITE DE POSICIONAMENTO AUTOMÁTICO DO SLIDE +PRZ03 OP120;1
   E0304 : BOOL ;	//=DCK_2++ZNE05+HCZ01-U_03;AVISO CARRO MOVIDRIVE +CRX01 - OP130;1
   E0305 : BOOL ;	//=DCK_2++ZNE05+HCZ01-U_04;AVISO MOVIDRIVE SLIDE +CRY01 - OP130;1
   E0306 : BOOL ;	//=DCK_2++ZNE05+HCZ01-U_06;AVISO MOVIDRIVE SLIDE +CRZ01 - OP130;1
   E0307 : BOOL ;	//=DCK_2++ZNE05+HCZ01-U_05;AVISO MOVIDRIVE SLIDE +CRY02 - OP130;1
   E0308 : BOOL ;	//=DCK_2++ZNE05+HCZ01-U_07;AVISO MOVIDRIVE SLIDE +CRZ02 - OP130;1
   E0309 : BOOL ;	//=DCK_2++ZNE05+HCZ01-U_08;AVISO MOVIDRIVE SLIDE +CRX02 - OP130;1
   E0310 : BOOL ;	//=DCK_2++ZNE05+HCZ01-U_09;AVISO MOVIDRIVE SLIDE +CRY03 - OP130;1
   E0311 : BOOL ;	//=DCK_2++ZNE05+HCZ01-U_11;AVISO MOVIDRIVE SLIDE +CRZ03 - OP130;1
   E0312 : BOOL ;	//=DCK_2++ZNE05+HCZ01-U_10;AVISO MOVIDRIVE SLIDE +CRY04 - OP130;1
   E0313 : BOOL ;	//=DCK_2++ZNE05+HCZ01-U_12;AVISO MOVIDRIVE SLIDE +CRZ04 - OP130;1
   E0314 : BOOL ;	//=DCK_2++ZNE05+HCZ01-U_16;AVISO PORTAL MOVIDRIVE +PRX01- OP120;1
   E0315 : BOOL ;	//=DCK_2++ZNE05+HCZ01-U_16;AVISO MOVIDRIVE SLIDE +PRZ01 - OP120;1
   E0316 : BOOL ;	//=DCK_2++ZNE05+HCZ01-U_16;AVISO MOVIDRIVE SLIDE +CRZ05 - OP130;1
   E0317 : BOOL ;	//=DCK_2++ZNE05+HCZ01-U_15;AVISO MOVIDRIVE SLIDE +PRZ02 - OP120;1
   E0318 : BOOL ;	//=DCK_2++ZNE05+HCZ01-U_17;AVISO MOVIDRIVE SLIDE +CRZ06 - OP130;1
   E0319 : BOOL ;	//=DCK_2++ZNE05+HCZ01-U_04;ANOMALIA DO PORTAL MOVIDRIVE +PRX02 - OP120;1
   E0320 : BOOL ;	//=DCK_2++ZNE05+CRZ02-SQ_01;SLIDE DE ALTA VIAGEM EXTRA +CRZ02 - OP130;1
   E0321 : BOOL ;	//=DCK_2++ZNE05+CRZ02-SQ_02;CODIFICADOR DE DESLIZAMENTO EXTRA BAIXO/ZERO +CRZ02 - OP130;1
   E0322 : BOOL ;	//=DCK_2++ZNE05+CRZ02-SQ_03;CHAVE DE FENDA EXTRA VIAGEM NO SLIDE +CRZ02 - OP130;1
   E0323 : BOOL ;	//=DCK_2++ZNE05+HCZ01-U_08;MOVIDRIVE SLIDE +CRX02 NÃO RESET - OP130;58
   E0324 : BOOL ;	//=DCK_2++ZNE05+HCZ01-U_08;ANOMALIA DO SLIDE MOVIDRIVE +CRX02 - OP130;1
   E0325 : BOOL ;	//=DCK_2++ZNE05+CRX02-SQ_01;TRANSPORTE DO CODIFICADOR REVERSO/ZERO DE VIAGEM EXTRA +CRX02-OP130;1
   E0326 : BOOL ;	//=DCK_2++ZNE05+CRX01-SQ_06;ANTICOL. ENTRE CARROS +CRX01 E +CRX02 BACK-UP-OP130;1
   E0327 : BOOL ;	//=DCK_2++ZNE05+HCZ01-U_09;MOVIDRIVE SLIDE +CRY03 NÃO RESET - OP130;58
   E0328 : BOOL ;	//=DCK_2++ZNE05+HCZ01-U_09;ANOMALIA DO SLIDE MOVIDRIVE +CRY03 - OP130;1
   E0329 : BOOL ;	//=DCK_2++ZNE05+CRY03-SQ_01;CODIFICADOR DE DESLIZAMENTO EXTRA/REVERSO DE VIAGEM ZERO CRY03-OP130;1
   E0330 : BOOL ;	//=DCK_2++ZNE05+CRY04-SQ_02;ANTICOLISÃO ENTRE SLIDES +CRY03 E +CRY04 - OP130;1
   E0331 : BOOL ;	//=DCK_2++ZNE05+HCZ01-U_11;ANOMALIA DO SLIDE MOVIDRIVE +CRZ03 - OP130;1
   E0332 : BOOL ;	//=DCK_2++ZNE05+CRZ03-SQ_01;SLIDE DE ALTA VIAGEM EXTRA +CRZ03 - OP130;1
   E0333 : BOOL ;	//=DCK_2++ZNE05+CRZ03-SQ_02;CODIFICADOR DE DESLIZAMENTO EXTRA BAIXO/ZERO +CRZ03 - OP130;1
   E0334 : BOOL ;	//=DCK_2++ZNE05+HCZ01-U_04;AVISO PORTAL MOVIDRIVE +PRX02 - OP120;1
   E0335 : BOOL ;	//=DCK_2++ZNE05+HCZ01-U_10;MOVIDRIVE SLIDE +CRY04 NÃO RESET - OP130;58
   E0336 : BOOL ;	//=DCK_2++ZNE05+HCZ01-QM_09;MAGN.INVERTER SLIDE + PARAFUSO CRY03. SX.+CRX02-OP130;1
   E0337 : BOOL ;	//=DCK_2++ZNE05+HCZ01-QF_48;DESLIZAMENTO DO MOTOR DE FREIO MAGN. +CRY03 PARAFUSO ESQUERDO.+CRX02-OP130;1
   E0338 : BOOL ;	//=DCK_2++ZNE05+HCZ01-QM_11;MAGN. INVERTIDO. DESLIZAMENTO + PARAFUSO CRZ03. SX.+CRX02 OP130;1
   E0339 : BOOL ;	//=DCK_2++ZNE05+HCZ01-QF_50;DESLIZAMENTO DO MOTOR DE FREIO MAGN. +CRZ03 PARAFUSO ESQUERDO.+CRX02 OP130;1
   E0340 : BOOL ;	//=DCK_2++ZNE05+HCZ01-QM_10;MAGN. INVERSOR DESLIZANTE +CRY04 PARAFUSAMENTO DIREITO+CRX02-OP130;1
   E0341 : BOOL ;	//=DCK_2++ZNE05+HCZ01-QF_49;DESLIZAMENTO DO MOTOR DE FREIO MAGN. + PARAFUSO DIREITO CRY04. + CRX02-OP130;1
   E0342 : BOOL ;	//=DCK_2++ZNE05+HCZ01-QM_12;MAGN.INVERTER SLIDE + PARAFUSO CRZ04. DX.+CRX02-OP130;1
   E0343 : BOOL ;	//=DCK_2++ZNE05+HCZ01-QF_51;DESLIZAMENTO DO MOTOR DE FREIO MAGN. +CRZ04 PARAFUSO DIREITO.+CRX02-OP130;1
   E0344 : BOOL ;	//=DCK_2++ZNE05+HCZ01-QM_15;MAGN. INVERSOR DE MOTOR TRADUÇÃO DE PORTAL +PRX01 - OP120;1
   E0345 : BOOL ;	//=DCK_2++ZNE05+HCZ01-QF_54;PORTAL TRADUÇÃO MOTOR FREIO MAGN +PRX01 OP120;1
   E0346 : BOOL ;	//=DCK_2++ZNE05+HCZ01-QM_16;MAGN.INVERSOR SLIDE +PRZ01 PARAFUSO ESQUERDO.+PRX01-OP120;1
   E0347 : BOOL ;	//=DCK_2++ZNE05+HCZ01-QF_55;DESLIZAMENTO DO MOTOR DE FREIO MAGN. +PRZ01 PARAFUSO ESQUERDO.+PRX01-OP120;1
   E0348 : BOOL ;	//=DCK_2++ZNE05+HCZ01-QM_13;MAGN.INVERTER SLIDE +CRZ05 ESQUERDA BASCU.+CRX02-OP130;1
   E0349 : BOOL ;	//=DCK_2++ZNE05+HCZ01-QF_52;MAGN.FREIO MOT.SLIDE +CRZ05 ESQUERDA BASCU.+CRX02-OP130;1
   E0350 : BOOL ;	//=DCK_2++ZNE05+HCZ01-QM_17;MAGN.INVERSOR SLIDE +PRZ02 PARAFUSO DIREITO.-OP120;1
   E0351 : BOOL ;	//=DCK_2++ZNE05+HCZ01-QF_56;MAGN.BRAKE MOTOR SLIDE +PRZ02 PARAFUSO DIREITO.-OP120;1
   E0352 : BOOL ;	//=DCK_2++ZNE05+HCZ01-U_10;ANOMALIA DO SLIDE MOVIDRIVE +CRY04 - OP130;1
   E0353 : BOOL ;	//=DCK_2++ZNE05+CRY04-SQ_01;EXTRA VIAGEM REVERSA/ZERO ENCODER SLIDE+CRY04 OP130;1
   E0354 : BOOL ;	//=DCK_2++ZNE05+CRY04-SQ_02;ANTICOLISÃO ENTRE SLIDES +CRY03 E +CRY04 - OP130;1
   E0355 : BOOL ;	//=DCK_2++ZNE05+HCZ01-U_12;ANOMALIA DO SLIDE MOVIDRIVE +CRZ04 - OP130;1
   E0356 : BOOL ;	//=DCK_2++ZNE05+CRZ04-SQ_01;SLIDE DE ALTA VIAGEM EXTRA +CRZ04 - OP130;1
   E0357 : BOOL ;	//=DCK_2++ZNE05+CRZ04-SQ_02;CODIFICADOR DE DESLIZAMENTO EXTRA BAIXO/ZERO +CRZ04 - OP130;1
   E0358 : BOOL ;	//=DCK_2++ZNE05+CRZ04-SQ_03;CHAVE DE FENDA EXTRA VIAGEM NO SLIDE +CRZ04 - OP130;1
   E0359 : BOOL ;	//=DCK_2++ZNE05+HCZ01-U_16;PORTAL MOVIDRIVE +PRX01 NÃO ZERO - OP120;1
   E0360 : BOOL ;	//=DCK_2++ZNE05+HCZ01-U_16;ANOMALIA DO PORTAL MOVIDRIVE +PRX01 - OP120;1
   E0361 : BOOL ;	//=DCK_2++ZNE05+PRX01-SQ_01;CODIFICADOR EXTRA VIAGEM VOLTA/ZERO PORTAL+PRX01-OP120;1
   E0362 : BOOL ;	//=DCK_2++ZNE05+PRX01-SQ_02;PORTAL AVANÇO VIAGEM EXTRA +PRX01-OP120;1
   E0363 : BOOL ;	//=DCK_2++ZNE05+HCZ01-U_16;MOVIDRIVE SLIDE +PRZ01 NÃO RESET - OP120;1
   E0364 : BOOL ;	//=DCK_2++ZNE05+HCZ01-U_14;ANOMALIA DO SLIDE MOVIDRIVE +PRZ01 - OP120;1
   E0365 : BOOL ;	//=DCK_2++ZNE05+PRZ01-SQ_01;DESLIZAMENTO DO CODIFICADOR EXTRA REVERSE/ZERO +PRZ01-OP120;1
   E0366 : BOOL ;	//=DCK_2++ZNE05+PRZ01-SQ_02;DESLIZAMENTO DO CODIFICADOR DE VIAGEM EXTRA PARA FRENTE +PRZ01-OP120;1
   E0367 : BOOL ;	//=DCK_2++ZNE05+HCZ01-U_16;ANOMALIA DO SLIDE MOVIDRIVE +CRZ05 - OP130;1
   E0368 : BOOL ;	//=DCK_2++ZNE05+CRZ05-SQ_01;SLIDE DE ALTA VIAGEM EXTRA +CRZ05 - OP130;1
   E0369 : BOOL ;	//=DCK_2++ZNE05+CRZ05-SQ_02;CODIFICADOR DE DESLIZAMENTO EXTRA BAIXO/ZERO +CRZ05 - OP130;1
   E0370 : BOOL ;	//=DCK_2++ZNE05;TRANSFERÊNCIAS DE ANOMALIA ENTRE ++ZNE04 --> ++ZNE08;1
   E0371 : BOOL ;	//=DCK_2++ZNE05+HCZ01-U_17;MOVIDRIVE SLIDE +PRZ02 NÃO RESET - OP120;58
   E0372 : BOOL ;	//=DCK_2++ZNE05+HCZ01-U_17;ANOMALIA DO SLIDE MOVIDRIVE +PRZ02 - OP120;1
   E0373 : BOOL ;	//=DCK_2++ZNE05+PRZ02-SQ_01;DESLIZAMENTO DO CODIFICADOR EXTRA REVERSE/ZERO+PRZ02-OP120;1
   E0374 : BOOL ;	//=DCK_2++ZNE05+PRZ02-SQ_04;SLIDE DE VIAGEM EXTRA PARA FRENTE +PRZ02 - OP120;1
   E0375 : BOOL ;	//=DCK_2++ZNE05+HCZ01-U_17;ANOMALIA DO SLIDE MOVIDRIVE +CRZ06 - OP130;1
   E0376 : BOOL ;	//=DCK_2++ZNE05+CRZ06-SQ_01;SLIDE DE ALTA VIAGEM EXTRA +CRZ06 - OP130;1
   E0377 : BOOL ;	//=DCK_2++ZNE05+CRZ06-SQ_02;SLIDE DO CODIFICADOR DE VIAGEM EXTRA BAIXO/ZERO +CRZ06 - OP130;1
   E0378 : BOOL ;
   E0379 : BOOL ;	//=DCK_2++ZNE05+CRX01-SQ_02;MANCATA POSIZIONE DI BACK-UP CARRO +CRX01 - OP130 ;58
   E0380 : BOOL ;	//=DCK_2++ZNE05+CRX02-SQ_02;MANCATA POSIZIONE DI BACK-UP CARRO +CRX02 - OP130 ;58
   E0381 : BOOL ;
   E0382 : BOOL ;	//=DCK_2++ZNE05+CRZ01-SQ_04;OBTURADOR DE SEGURANÇA +CRZ01 DISPARADO - OP130;1
   E0383 : BOOL ;	//=DCK_2++ZNE05+CRZ02-SQ_04;OBTURADOR DE SEGURANÇA +CRZ02 DISPARADO - OP130;1
   E0384 : BOOL ;	//=DCK_2++ZNE05+HCZ01-QM_14;MAGN.INVERTER SLIDE +CRZ06 DIREITA BASCU.+CRX02-OP130;1
   E0385 : BOOL ;	//=DCK_2++ZNE05+HCZ01-QF_53;MAGN.FREIO DESLIZANTE +CRZ06 DIREITA BASCU.+CRX02-OP130;1
   E0386 : BOOL ;	//=DCK_2++ZNE05+CRX01-SQ_01;TRANSPORTE DO CODIFICADOR REVERSO/ZERO DE VIAGEM EXTRA +CRX01-OP130;1
   E0387 : BOOL ;	//=DCK_2++ZNE05+SWK05-SWK05;SISTEMA DE CHAVE DE FENDA ATLAS NÃO PRONTO OP130 CRX03;58
   E0388 : BOOL ;	//=DCK_2++ZNE05+SWK05-SWK07;SISTEMA DE CHAVE DE FENDA ATLAS NÃO PRONTO OP130 CRX04 SX;58
   E0389 : BOOL ;	//=DCK_2++ZNE05+CRZ03-SQ_03;CHAVE DE FENDA EXTRA VIAGEM NO SLIDE +CRZ03 - OP130;1
   E0390 : BOOL ;	//=DCK_2++ZNE05+SWK06-SWK09;SISTEMA DE CHAVE DE FENDA ATLAS NÃO PRONTO OP130 CRX04 DX;58
   E0391 : BOOL ;
   E0392 : BOOL ;	//=DCK_2++ZNE05+HCZ01-QM_18;MAGN.INVERSOR SLIDE +PRZ03 PARAFUSO DIREITO.-OP120;1
   E0393 : BOOL ;	//=DCK_2++ZNE05+HCZ01-QF_57;MAGN.BRAKE MOTOR SLIDE +PRZ03 PARAFUSO DIREITO.-OP120;1
   E0394 : BOOL ;	//=DCK_2++ZNE05+HCZ01-U_18;MOVIDRIVE SLIDE +PRZ03 NÃO RESET - OP120;58
   E0395 : BOOL ;	//=DCK_2++ZNE05+HCZ01-U_18;ANOMALIA DO SLIDE MOVIDRIVE +PRZ03 - OP120;1
   E0396 : BOOL ;	//=DCK_2++ZNE05+PRZ03-SQ_01;DESLIZAMENTO DO CODIFICADOR EXTRA REVERSE/ZERO+PRZ03-OP120;1
   E0397 : BOOL ;	//=DCK_2++ZNE05+PRZ03-SQ_02;SLIDE DE VIAGEM EXTRA PARA FRENTE +PRZ03 - OP120;1
   E0398 : BOOL ;	//=DCK_2++ZNE05+HCZ01-U_18;AVISO MOVIDRIVE SLIDE +PRZ03 - OP120;1
   E0399 : BOOL ;
   E0400 : BOOL ;	//=DCK_2++ZNE05+CRZ03-SQ_04;OBTURADOR DE SEGURANÇA +CRZ03 DISPARADO - OP130;1
   E0401 : BOOL ;	//=DCK_2++ZNE05+CRZ04-SQ_04;OBTURADOR DE SEGURANÇA +CRZ04 DISPARADO - OP130;1
   E0402 : BOOL ;	//=DCK_2++ZNE05+PRZ01-SQ_04;OBTURADOR DE SEGURANÇA +PRZ01 DISPARADO - OP120;1
   E0403 : BOOL ;	//=DCK_2++ZNE05+PRZ02-SQ_07;OBTURADOR DE SEGURANÇA +PRZ02 DISPARADO - OP120;1
   E0404 : BOOL ;	//=DCK_2++ZNE05+PRZ03-SQ_07;OBTURADOR DE SEGURANÇA +PRZ03 DISPARADO - OP120;1
   E0405 : BOOL ;
   E0406 : BOOL ;	//=DCK_2++ZNE05+HKM05-DMC01;NÓ 38 PROFINET ET200S CAIXA MÓVEL CRX03 OP130;1
   E0407 : BOOL ;	//=DCK_2++ZNE05+HKM06-DMC01;NÓ 39 PROFINET ET200S CAIXA MÓVEL CRX04 OP130;1
   E0408 : BOOL ;	//=DCK_2++ZNE05+HKM01-DMC01;NÓ 30 PROFINET ET200S CAIXA FIXA OP130;1
   E0409 : BOOL ;	//=DCK_2++ZNE05+HKM02-DMC01;NÓ 31 PROFINET ET200S CAIXA MÓVEL CRX01 OP130;1
   E0410 : BOOL ;	//=DCK_2++ZNE05+HKM03-DMC01;NÓ 33 PROFINET ET200S CAIXA MÓVEL CRX02 OP130;1
   E0411 : BOOL ;	//=DCK_2++ZNE05+HKM04-DMC01;NÓ 34 PROFINET ET200S CAIXA MÓVEL PRX01 OP120;1
   E0412 : BOOL ;	//=DCK_2++ZNE05+HCZ01-A__04;CARTÃO NODE 90 PROFINET UFR41B SEW OP130;1
   E0413 : BOOL ;	//=DCK_2++ZNE05+HCZ01-A__02;NÓ 91 PROFINET UFR41B PLACA COSTURA OP120/OP130;1
   E0414 : BOOL ;	//=DCK_2++ZNE05+HCZ01-A__03;CARTÃO NODE 92 PROFINET UFR41B SEW OP130;1
   E0415 : BOOL ;	//=DCK_2++ZNE05+SWK01-SWK01;NODE 160 CHAVES DE FENDA PROFINET ATLAS OP120 SX.;58
   E0416 : BOOL ;	//=DCK_2++ZNE05+SWK01-SWK03;NODE 161 CHAVES DE FENDA PROFINET ATLAS OP120 SX.;58
   E0417 : BOOL ;	//=DCK_2++ZNE05+SWK02-SWK06;NODE 162 CHAVES DE FENDA PROFINET ATLAS OP120 DX.;58
   E0418 : BOOL ;	//=DCK_2++ZNE05+SWK02-SWK08;NODE 163 CHAVES DE FENDA PROFINET ATLAS OP120 DX.;58
   E0419 : BOOL ;	//=DCK_2++ZNE05+SWK03-SWK01;NODE 164 CHAVES DE FENDA PROFINET ATLAS OP130 SX.CRX02;58
   E0420 : BOOL ;	//=DCK_2++ZNE05+SWK04-SWK03;NODE 165 CHAVES DE FENDA PROFINET ATLAS OP130 DX.CRX01;58
   E0421 : BOOL ;	//=DCK_2++ZNE05+SWK05-SWK05;NODE 166 CHAVES DE FENDA PROFINET ATLAS OP130 SX.CRX03;58
   E0422 : BOOL ;	//=DCK_2++ZNE05+SWK05-SWK07;NODE 167 CHAVES DE FENDA PROFINET ATLAS OP130 SX.CRX04;58
   E0423 : BOOL ;	//=DCK_2++ZNE05+SWK06-SWK09;NODE 168 CHAVES DE FENDA PROFINET ATLAS OP130 DX.CRX04;58
   E0424 : BOOL ;	//=DCK_2++ZNE05+CRX01;BACK-UP AUTOMÁTICO CARRO1 (PARAFUSOS COM CARRO3);55
   E0425 : BOOL ;	//=DCK_2++ZNE05+CRX02;BACK-UP AUTOMÁTICO CARRO2 (PARAFUSOS COM CARRO4 OP135);55
   E0426 : BOOL ;	//=DCK_2++ZNE05+CRX03;BACK-UP AUTOMÁTICO CARRO3 (PARAFUSOS COM CARRO1 OP135);55
   E0427 : BOOL ;	//=DCK_2++ZNE05+SWK01-SWK01;SISTEMA DE CHAVE DE FENDA ATLAS NÃO ESTÁ PRONTO OP120 SX;58
   E0428 : BOOL ;	//=DCK_2++ZNE05+SWK01-SWK03;SISTEMA DE CHAVE DE FENDA ATLAS NÃO ESTÁ PRONTO OP120 SX;58
   E0429 : BOOL ;	//=DCK_2++ZNE05+SWK02-SWK06;SISTEMA DE CHAVE DE FENDA ATLAS NÃO PRONTO OP120 DX;58
   E0430 : BOOL ;	//=DCK_2++ZNE05+SWK02-SWK08;SISTEMA DE CHAVE DE FENDA ATLAS NÃO PRONTO OP120 DX;58
   E0431 : BOOL ;	//=DCK_2++ZNE05+SWK03-SWK01;SISTEMA DE CHAVE DE FENDA ATLAS NÃO PRONTO OP130 CRX02;58
   E0432 : BOOL ;	//=DCK_2++ZNE05+SWK04-SWK03;SISTEMA DE CHAVE DE FENDA ATLAS NÃO PRONTO OP130 CRX01;58
   E0433 : BOOL ;	//=DCK_2++ZNE05+CRX01-SQ_02;POSIÇÃO FALTA. CARRO DE BACK-UP CORRETO +CRX01-OP130;58
   E0434 : BOOL ;	//=DCK_2++ZNE05+CRX02-SQ_02;POSIÇÃO FALTA. CARRO DE BACK-UP CORRETO +CRX02-OP130;58
   E0435 : BOOL ;	//=DCK_2++ZNE05+CRX04;BACK-UP AUTOMÁTICO CARRO4 (PARAFUSOS COM CARRO2 OP135);55
   E0436 : BOOL ;	//=DCK_2++ZNE05+CRX01-SQ_03; POSIZIONE BARRA PUFFER ERRATA +CRX01-OP130;1
   E0437 : BOOL ;	//=DCK_2++ZNE05+CRX01-SQ_04; POSIZIONE BARRA PUFFER BACKUP ERRATA +CRX01-OP130;1
   E0438 : BOOL ;	//=DCK_2++ZNE05+CRX02-SQ_03; POSIZIONE BARRA PUFFER ERRATA +CRX02-OP130;1
   E0439 : BOOL ;	//=DCK_2++ZNE05+CRX02-SQ_04; POSIZIONE BARRA PUFFER BACKUP ERRATA +CRX02-OP130;1
   E0440 : BOOL ;	//=DCK_2++ZNE05+PRZ01;SLIDE +PRZ01 DESATIVADO OP120;55
   E0441 : BOOL ;	//=DCK_2++ZNE05+PRZ02;SLIDE +PRZ02 DESATIVADO OP120;55
   E0442 : BOOL ;	//=DCK_2++ZNE05+PRZ03;SLIDE +PRZ03 DESATIVADO OP120;55
   E0443 : BOOL ;	//=DCK_2++ZNE05+PRZ04;SLIDE +PRZ04 DESATIVADO OP120;55
   E0444 : BOOL ;	//=DCK_2++ZNE05+SWK02-SWK10;NODE 87 CHAVES DE FENDA PROFINET ATLAS OP120 DX;58
   E0445 : BOOL ;	//=DCK_2++ZNE05+SWK02-SWK10;SISTEMA DE CHAVE DE FENDA ATLAS NÃO PRONTO OP120 DX;58
   E0446 : BOOL ;
   E0447 : BOOL ;
   E0448 : BOOL ;	//=DCK_2++ZNE05;COMANDO DE ENVIO OP120 FALTA NO NPL MES;58
   E0449 : BOOL ;	//=DCK_2++ZNE05;COMANDO DE ENVIO OP130 FALTA NO NPL MES;58
   E0450 : BOOL ;	//=DCK_2++ZNE05+TR_01;BYPASS PRÉ-ALARME ATIVO EM +TR_01-OP120;54
   E0451 : BOOL ;	//=DCK_2++ZNE05+TR_02;BYPASS PRÉ-ALARME ATIVO EM +TR_02-OP130;54
   E0452 : BOOL ;	//=DCK_2++ZNE05;PRÉ-ALARME ++ZNE05 EM CICLO DE MANUTENÇÃO;13
   E0453 : BOOL ;
   E0454 : BOOL ;
   E0455 : BOOL ;
   E0456 : BOOL ;	//=DCK_2++ZNE05+HCZ01-QM_27;SLIDE MAGN. +CRZ09 PARAFUSO INTERNO ESQUERDO EM +CRX04;1
   E0457 : BOOL ;	//=DCK_2++ZNE05+HCZ01-QM_28;SLIDE MAGN. +CRZ10 CHAVE DE FENDA INTERNA DIREITA EM +CRX04;1
   E0458 : BOOL ;	//=DCK_2++ZNE05+HCZ01-QM_29;SLIDE MAGN. +CRZ11 PARAFUSO EXTERNO ESQUERDO EM +CRX04;1
   E0459 : BOOL ;	//=DCK_2++ZNE05+HCZ01-QM_30;SLIDE MAGN. +CRZ12 CHAVE DE FENDA EXTERNA DIREITA EM +CRX04;1
   E0460 : BOOL ;	//=DCK_2++ZNE05+HCZ01-QM_25;SLIDE MAGN. +CRY07 CHAVE DE FENDA ESQUERDA EM +CRX04 OP130;1
   E0461 : BOOL ;	//=DCK_2++ZNE05+HCZ01-QM_26;SLIDE MAGN. +CRY08 CHAVE DE FENDA DIREITA EM +CRX04 OP130;1
   E0462 : BOOL ;	//=DCK_2++ZNE05+HCZ01-QF_26;CARRO INVERSOR DE ALIMENTAÇÃO MAGN. +CRX03;1
   E0463 : BOOL ;	//=DCK_2++ZNE05+HCZ01-QF_87;CARRO INVERSOR DE ALIMENTAÇÃO MAGN. +CRX04;1
   E0464 : BOOL ;	//=DCK_2++ZNE05+HCZ01-QF_61;MAGN.BRAKE SLIDE +CRZ07 CHAVE DE FENDA ESQUERDA +CRX03;1
   E0465 : BOOL ;	//=DCK_2++ZNE05+HCZ01-QF_62;MAGN.BRAKE SLIDE +CRZ08 CHAVE DE FENDA PARA CIMA +CRX03;1
   E0466 : BOOL ;	//=DCK_2++ZNE05+HCZ01-QF_66;MAGN.BRAKE SLIDE +CRZ09 PARAFUSO INTERNO ESQUERDO ON +CRX04;1
   E0467 : BOOL ;	//=DCK_2++ZNE05+HCZ01-QF_67;MAGN.BRAKE SLIDE +CRZ10 PARAFUSO INTERNO DIREITO EM +CRX04;1
   E0468 : BOOL ;	//=DCK_2++ZNE05+HCZ01-QF_68;MAGN.BRAKE SLIDE +CRZ11 PARAFUSO EXTERNO ESQUERDO ON +CRX04;1
   E0469 : BOOL ;	//=DCK_2++ZNE05+HCZ01-QF_69;MAGN.BRAKE SLIDE +CRZ12 PARAFUSO EXTERNO DIREITO EM +CRX04;1
   E0470 : BOOL ;	//=DCK_2++ZNE05+HCZ01-QM_20;SLIDE MAGN. +CRY05 CHAVE DE FENDA ESQUERDA NO CARRO +CRX03;1
   E0471 : BOOL ;	//=DCK_2++ZNE05+HCZ01-QM_21;MAGN.SLIDE +CRY06 CHAVE DE FENDA DIREITA NO CARRO +CRX03;1
   E0472 : BOOL ;	//=DCK_2++ZNE05+HCZ01-QM_22;SLIDE MAGN. +CRZ07 CHAVE DE FENDA ESQUERDA NO CARRO +CRX03;1
   E0473 : BOOL ;	//=DCK_2++ZNE05+HCZ01-QM_19;MOTOR DE TRADUÇÃO DE CARRO MAGN.INVERTER +CRX03;1
   E0474 : BOOL ;	//=DCK_2++ZNE05+HCZ01-ST_08;RESISTOR DE FREIO DE TRADUÇÃO DE CARRO +CRX03;1
   E0475 : BOOL ;	//=DCK_2++ZNE05+HCZ01-QM_23;MAGN.SLIDE +CRZ08 CHAVE DE FENDA DIREITA NO CARRO +CRX03;1
   E0476 : BOOL ;	//=DCK_2++ZNE05+HCZ01-ST_09;RESISTOR DE FREIO DE TRADUÇÃO DE CARRO +CRX04;1
   E0477 : BOOL ;	//=DCK_2++ZNE05+HCZ01-QM_24;MOTOR DE TRADUÇÃO DE CARRO MAGN.INVERTER +CRX04;1
   E0478 : BOOL ;	//=DCK_2++ZNE05+HCZ01-QF_58;CARRO DE TRADUÇÃO MOTOR MAGN.BRAKE +CRX03 OP.130;1
   E0479 : BOOL ;	//=DCK_2++ZNE05+HCZ01-QF_59;MAGN.BRAKE SLIDE +CRY05 CHAVE DE FENDA ESQUERDA EM +CRX03;1
   E0480 : BOOL ;	//=DCK_2++ZNE05+HCZ01-QF_60;MAGN.BRAKE SLIDE +CRY06 CHAVE DE FENDA DIREITA EM +CRX03;1
   E0481 : BOOL ;	//=DCK_2++ZNE05+HCZ01-QF_63;CARRO DE TRADUÇÃO DO MOTOR MAGN.BRAKE +CRX04 OP.130;1
   E0482 : BOOL ;	//=DCK_2++ZNE05+HCZ01-QF_64;MAGN.BRAKE SLIDE +CRY07 CHAVE DE FENDA ESQUERDA LIGADA +CRX04;1
   E0483 : BOOL ;	//=DCK_2++ZNE05+HCZ01-QF_65;MAGN.BRAKE SLIDE +CRY08 CHAVE DE FENDA DIREITA EM +CRX04;1
   E0484 : BOOL ;	//=DCK_2++ZNE05+HCZ01-ST_03;RESISTÊNCIA À TRAVAGEM DE TRADUÇÃO +CRX01 OP130;1
   E0485 : BOOL ;	//=DCK_2++ZNE05+HCZ01-ST_04;RESISTÊNCIA À TRAVAGEM DE TRADUÇÃO +CRX02 OP130;1
   E0486 : BOOL ;
   E0487 : BOOL ;
   E0488 : BOOL ;	//=DCK_2++ZNE05+HCZ01-KA_30;SÉRIE FEEDBACK HABILITA MOVIDRIVE EIXO Z +CRZ07;2
   E0489 : BOOL ;	//=DCK_2++ZNE05+HCZ01-KA_31;SÉRIE FEEDBACK HABILITA MOVIDRIVE EIXO Z +CRZ08;2
   E0490 : BOOL ;	//=DCK_2++ZNE05+HCZ01-KA_32;SÉRIE FEEDBACK HABILITA MOVIDRIVE EIXO X +CRX04;2
   E0491 : BOOL ;	//=DCK_2++ZNE05+HCZ01-KA_33;SÉRIE FEEDBACK HABILITA MOVIDRIVE EIXO Y +CRY07/+CRY08;2
   E0492 : BOOL ;	//=DCK_2++ZNE05+HCZ01-KA_34;SÉRIE FEEDBACK HABILITA MOVIDRIVE EIXO Z +CRZ09;2
   E0493 : BOOL ;	//=DCK_2++ZNE05+HCZ01-KA_35;SÉRIE FEEDBACK HABILITA MOVIDRIVE EIXO Z +CRZ10;2
   E0494 : BOOL ;	//=DCK_2++ZNE05+HCZ01-KA_28;SÉRIE FEEDBACK HABILITA MOVIDRIVE EIXO X +CRX03;2
   E0495 : BOOL ;	//=DCK_2++ZNE05+HCZ01-KA_29;SÉRIE FEEDBACK HABILITA MOVIDRIVE EIXO Y +CRY05/+CRY06;2
   E0496 : BOOL ;	//=DCK_2++ZNE05+HCZ01-KA_36;SÉRIE FEEDBACK HABILITA MOVIDRIVE EIXO Z +CRZ11;2
   E0497 : BOOL ;	//=DCK_2++ZNE05+HCZ01-KA_37;SÉRIE FEEDBACK HABILITA MOVIDRIVE EIXO Z +CRZ12;2
   E0498 : BOOL ;
   E0499 : BOOL ;
   E0500 : BOOL ;
   E0501 : BOOL ;
   E0502 : BOOL ;
   E0503 : BOOL ;
   E0504 : BOOL ;	//=DCK_2++ZNE05+CRZ07-SQ_03;CHAVE DE FENDA EXTRA DE VIAGEM NO SLIDE +CRZ07;1
   E0505 : BOOL ;	//=DCK_2++ZNE05+CRZ08-SQ_03;CHAVE DE FENDA EXTRA DE VIAGEM NO SLIDE +CRZ08;1
   E0506 : BOOL ;	//=DCK_2++ZNE05+CRZ09-SQ_03;CHAVE DE FENDA EXTRA DE VIAGEM NO SLIDE +CRZ09;1
   E0507 : BOOL ;	//=DCK_2++ZNE05+CRZ10-SQ_03;CHAVE DE FENDA EXTRA DE VIAGEM NO SLIDE +CRZ10;1
   E0508 : BOOL ;	//=DCK_2++ZNE05+CRZ11-SQ_03;CHAVE DE FENDA EXTRA DE VIAGEM NO SLIDE +CRZ11;1
   E0509 : BOOL ;	//=DCK_2++ZNE05+CRZ12-SQ_03;CHAVE DE FENDA EXTRA DE VIAGEM NO SLIDE +CRZ12;1
   E0510 : BOOL ;	//=DCK_2++ZNE05+CRX03-SQ_01;VIAGEM EXTRA PARA TRÁS NO CARRO +CRX03;1
   E0511 : BOOL ;	//=DCK_2++ZNE05+CRX04-SQ_01;VIAGEM EXTRA PARA TRÁS NO CARRO +CRX04;1
   E0512 : BOOL ;	//=DCK_2++ZNE05+CRY05-SQ_01;VIAGEM EXTRA PARA TRÁS NO SLIDE +CRY05;1
   E0513 : BOOL ;	//=DCK_2++ZNE05+CRY06-SQ_01;VIAGEM EXTRA PARA TRÁS NO SLIDE +CRY06;1
   E0514 : BOOL ;	//=DCK_2++ZNE05+CRY07-SQ_01;VIAGEM EXTRA PARA TRÁS NO SLIDE +CRY07;1
   E0515 : BOOL ;	//=DCK_2++ZNE05+CRY08-SQ_01;VIAGEM EXTRA PARA TRÁS NO SLIDE +CRY08;1
   E0516 : BOOL ;	//=DCK_2++ZNE05+CRZ07-SQ_01;ALTA VIAGEM EXTRA NO SLIDE +CRZ07;1
   E0517 : BOOL ;	//=DCK_2++ZNE05+CRZ07-SQ_02;BAIXA VIAGEM EXTRA NO SLIDE +CRZ07;1
   E0518 : BOOL ;	//=DCK_2++ZNE05+CRZ08-SQ_01;ALTA VIAGEM EXTRA NO SLIDE +CRZ08;1
   E0519 : BOOL ;	//=DCK_2++ZNE05+CRZ08-SQ_02;BAIXA VIAGEM EXTRA NO SLIDE +CRZ08;1
   E0520 : BOOL ;	//=DCK_2++ZNE05+CRZ09-SQ_01;ALTA VIAGEM EXTRA NO SLIDE +CRZ09;1
   E0521 : BOOL ;	//=DCK_2++ZNE05+CRZ09-SQ_02;BAIXA VIAGEM EXTRA NO SLIDE +CRZ09;1
   E0522 : BOOL ;	//=DCK_2++ZNE05+CRZ10-SQ_01;ALTA VIAGEM EXTRA NO SLIDE +CRZ10;1
   E0523 : BOOL ;	//=DCK_2++ZNE05+CRZ10-SQ_02;BAIXA VIAGEM EXTRA NO SLIDE +CRZ10;1
   E0524 : BOOL ;	//=DCK_2++ZNE05+CRZ11-SQ_01;ALTA VIAGEM EXTRA NO SLIDE +CRZ11;1
   E0525 : BOOL ;	//=DCK_2++ZNE05+CRZ11-SQ_02;BAIXA VIAGEM EXTRA NO SLIDE +CRZ11;1
   E0526 : BOOL ;	//=DCK_2++ZNE05+CRZ12-SQ_01;ALTA VIAGEM EXTRA NO SLIDE +CRZ12;1
   E0527 : BOOL ;	//=DCK_2++ZNE05+CRZ12-SQ_02;BAIXA VIAGEM EXTRA NO SLIDE +CRZ12;1
   E0528 : BOOL ;	//=DCK_2++ZNE05+CRX01-SQ_05;ANTICOLLISÃO ENTRE CARROS +CRX01 E +CRX03;1
   E0529 : BOOL ;	//=DCK_2++ZNE05+CRX01-SQ_06;ANTICOL. ENTRE CARROS DE BACK-UP +CRX01 E +CRX03;1
   E0530 : BOOL ;	//=DCK_2++ZNE05+CRX02-SQ_04;ANTICOLLISÃO ENTRE CARROS +CRX04 E +CRX02;1
   E0531 : BOOL ;	//=DCK_2++ZNE05+CRX04-SQ_05;ANTICOLLISÃO ENTRE CARREGAMENTOS +CRX03 E +CRX04;1
   E0532 : BOOL ;	//=DCK_2++ZNE05+CRX04-SQ_06;ANTICOL. ENTRE CARROS DE BACK-UP +CRX03 E +CRX04;1
   E0533 : BOOL ;	//=DCK_2++ZNE05+CRY05-SQ_02;ANTICOLISÃO ENTRE OS SLIDES +CRY05 E +CRY06;1
   E0534 : BOOL ;	//=DCK_2++ZNE05+CRY08-SQ_02;ANTICOLISÃO ENTRE OS SLIDES +CRY07 E +CRY08;1
   E0535 : BOOL ;
   E0536 : BOOL ;	//=DCK_2++ZNE05+TR_01-SE_02;FALHA NO NÓ 140 PROFISSIONAL ANTICOLISÃO TRASEIRO -SE_02;1
   E0537 : BOOL ;	//=DCK_2++ZNE05+TR_01-SE_03;FALHA NO NÓ 141 PROFISSIONAL ANTICOLISÃO DIANTEIRO -SE_03;1
   E0538 : BOOL ;	//=DCK_2++ZNE05+TR_02-SE_02;FALHA NO NÓ 142 PROFISSIONAL ANTICOLISÃO TRASEIRO -SE_02;1
   E0539 : BOOL ;	//=DCK_2++ZNE05+TR_02-SE_03;FALHA NO NÓ 143 ANTICOLISÃO DIANTEIRA PROF.;1
   E0540 : BOOL ;	//=DCK_2++ZNE05+TR_01-U__01;NÓ 124 ROLOS INVERSORES PROFINET +TR_01;1
   E0541 : BOOL ;	//=DCK_2++ZNE05+TR_02-U__02;ROLOS INVERSORES PROFINET NODE 125 +TR_02;1
   E0542 : BOOL ;
   E0543 : BOOL ;
   E0544 : BOOL ;	//=DCK_2++ZNE05+CRZ07-SQ_04;OBTURADOR DE SEGURANÇA +CRZ07 DISPARADO - OP130;1
   E0545 : BOOL ;	//=DCK_2++ZNE05+CRZ08-SQ_04;OBTURADOR DE SEGURANÇA +CRZ08 DISPARADO - OP130;1
   E0546 : BOOL ;	//=DCK_2++ZNE05+CRZ09-SQ_04;OBTURADOR DE SEGURANÇA +CRZ09 DISPARADO - OP130;1
   E0547 : BOOL ;	//=DCK_2++ZNE05+CRZ10-SQ_04;OBTURADOR DE SEGURANÇA +CRZ10 DISPARADO - OP130;1
   E0548 : BOOL ;	//=DCK_2++ZNE05+CRZ11-SQ_04;OBTURADOR DE SEGURANÇA +CRZ11 DISPARADO - OP130;1
   E0549 : BOOL ;	//=DCK_2++ZNE05+CRZ12-SQ_04;OBTURADOR DE SEGURANÇA +CRZ12 DISPARADO - OP130;1
   E0550 : BOOL ;
   E0551 : BOOL ;
   E0552 : BOOL ;	//=DCK_2++ZNE05+CRX03-SQ_02;FALHA NA POSIÇÃO DE RESERVA DO CARRO +CRX03 - OP130;58
   E0553 : BOOL ;	//=DCK_2++ZNE05+CRX04-SQ_02;FALHA NA POSIÇÃO DE RESERVA DO CARRO +CRX04 - OP130;58
   E0554 : BOOL ;
   E0555 : BOOL ;
   E0556 : BOOL ;
   E0557 : BOOL ;
   E0558 : BOOL ;
   E0559 : BOOL ;
   E0560 : BOOL ;	//=DCK_2++ZNE05+CRX01-SQ_04;POSIÇÃO ERRADA DA BARRA DO PUFFER DE BACKUP +CRX01-OP130;1
   E0561 : BOOL ;	//=DCK_2++ZNE05+CRX03-SQ_04;POSIÇÃO ERRADA DA BARRA DO PUFFER DE BACKUP +CRX03-OP130;1
   E0562 : BOOL ;	//=DCK_2++ZNE05+CRX04-SQ_04;POSIÇÃO ERRADA DA BARRA DO PUFFER DE BACKUP +CRX04-OP130;1
   E0563 : BOOL ;	//=DCK_2++ZNE05+CRX03-SQ_03;POSIÇÃO ERRADA DA BARRA DO PUFFER +CRX03-OP130;1
   E0564 : BOOL ;	//=DCK_2++ZNE05+CRX04-SQ_03;POSIÇÃO ERRADA DA BARRA DO PUFFER +CRX04-OP130;1
   E0565 : BOOL ;
   E0566 : BOOL ;
   E0567 : BOOL ;
   E0568 : BOOL ;	//=DCK_2++ZNE05+HCZ01-U_19;AVISO CARRO MOVIDRIVE +CRX03 - OP130;1
   E0569 : BOOL ;	//=DCK_2++ZNE05+HCZ01-U_20;AVISO MOVIDRIVE SLIDE +CRY05 - OP130;1
   E0570 : BOOL ;	//=DCK_2++ZNE05+HCZ01-U_21;AVISO MOVIDRIVE SLIDE +CRY06 - OP130;1
   E0571 : BOOL ;	//=DCK_2++ZNE05+HCZ01-U_22;AVISO MOVIDRIVE SLIDE +CRZ07 - OP130;1
   E0572 : BOOL ;	//=DCK_2++ZNE05+HCZ01-U_23;AVISO MOVIDRIVE SLIDE +CRZ08 - OP130;1
   E0573 : BOOL ;	//=DCK_2++ZNE05+HCZ01-U_24;AVISO CARRO MOVIDRIVE +CRX04 - OP130;1
   E0574 : BOOL ;	//=DCK_2++ZNE05+HCZ01-U_25;AVISO MOVIDRIVE SLIDE +CRY07 - OP130;1
   E0575 : BOOL ;	//=DCK_2++ZNE05+HCZ01-U_26;AVISO MOVIDRIVE SLIDE +CRY08 - OP130;1
   E0576 : BOOL ;	//=DCK_2++ZNE05+HCZ01-U_27;AVISO MOVIDRIVE SLIDE +CRZ09 - OP130;1
   E0577 : BOOL ;	//=DCK_2++ZNE05+HCZ01-U_28;AVISO MOVIDRIVE SLIDE +CRZ10 - OP130;1
   E0578 : BOOL ;	//=DCK_2++ZNE05+HCZ01-U_29;AVISO MOVIDRIVE SLIDE +CRZ11 - OP130;1
   E0579 : BOOL ;	//=DCK_2++ZNE05+HCZ01-U_30;AVISO MOVIDRIVE SLIDE +CRZ12 - OP130;1
   E0580 : BOOL ;
   E0581 : BOOL ;
   E0582 : BOOL ;
   E0583 : BOOL ;
   E0584 : BOOL ;	//=DCK_2++ZNE05+HCZ01-U_19;CARRO MOVIDRIVE +CRX03 NÃO RESET - OP130;58
   E0585 : BOOL ;	//=DCK_2++ZNE05+HCZ01-U_20;MOVIDRIVE SLIDE +CRY05 NÃO RESET - OP130;58
   E0586 : BOOL ;	//=DCK_2++ZNE05+HCZ01-U_21;MOVIDRIVE SLIDE +CRY06 NÃO RESET - OP130;58
   E0587 : BOOL ;	//=DCK_2++ZNE05+HCZ01-U_22;MOVIDRIVE SLIDE +CRZ07 NÃO RESET - OP130;58
   E0588 : BOOL ;	//=DCK_2++ZNE05+HCZ01-U_23;MOVIDRIVE SLIDE +CRZ08 NÃO RESET - OP130;58
   E0589 : BOOL ;	//=DCK_2++ZNE05+HCZ01-U_24;CARRO MOVIDRIVE +CRX04 NÃO RESET - OP130;58
   E0590 : BOOL ;	//=DCK_2++ZNE05+HCZ01-U_25;MOVIDRIVE SLIDE +CRY07 NÃO RESET - OP130;58
   E0591 : BOOL ;	//=DCK_2++ZNE05+HCZ01-U_26;MOVIDRIVE SLIDE +CRY08 NÃO REINICIALIZADO - OP130;58
   E0592 : BOOL ;	//=DCK_2++ZNE05+HCZ01-U_27;MOVIDRIVE SLIDE +CRZ09 NÃO RESET - OP130;58
   E0593 : BOOL ;	//=DCK_2++ZNE05+HCZ01-U_28;MOVIDRIVE SLIDE +CRZ10 NÃO RESET - OP130;58
   E0594 : BOOL ;	//=DCK_2++ZNE05+HCZ01-U_29;MOVIDRIVE SLIDE +CRZ11 NÃO RESET - OP130;58
   E0595 : BOOL ;	//=DCK_2++ZNE05+HCZ01-U_30;MOVIDRIVE SLIDE +CRZ12 NÃO RESET - OP130;58
   E0596 : BOOL ;	//=DCK_2++ZNE05+HCZ01-U_30;PORTAL MOVIDRIVE +PRX02 NÃO ZERO - OP120;58
   E0597 : BOOL ;
   E0598 : BOOL ;
   E0599 : BOOL ;
   E0600 : BOOL ;	//=DCK_2++ZNE05+CRX03;POSICIONAMENTO DO CARRO TIME-OUT +CRX03 OP130;1
   E0601 : BOOL ;	//=DCK_2++ZNE05+CRY05;TEMPO LIMITE DE POSICIONAMENTO AUTOMÁTICO DO SLIDE +CRY05 OP130;1
   E0602 : BOOL ;	//=DCK_2++ZNE05+CRY06;TEMPO LIMITE DE POSICIONAMENTO AUTOMÁTICO DO SLIDE +CRY06 OP130;1
   E0603 : BOOL ;	//=DCK_2++ZNE05+CRZ07;TEMPO LIMITE DE POSICIONAMENTO AUTOMÁTICO DO SLIDE +CRZ07 OP130;1
   E0604 : BOOL ;	//=DCK_2++ZNE05+CRZ08;TEMPO LIMITE DE POSICIONAMENTO AUTOMÁTICO DO SLIDE +CRZ08 OP130;1
   E0605 : BOOL ;	//=DCK_2++ZNE05+CRX04;POSICIONAMENTO DO CARRO TIME-OUT +CRX04 OP130;1
   E0606 : BOOL ;	//=DCK_2++ZNE05+CRY07;POSICIONAMENTO AUTOMÁTICO DO SLIDE TIME-OUT +CRY07 OP130;1
   E0607 : BOOL ;	//=DCK_2++ZNE05+CRY08;POSICIONAMENTO AUTOMÁTICO DO SLIDE TIME-OUT +CRY08 OP130;1
   E0608 : BOOL ;	//=DCK_2++ZNE05+CRZ09;TEMPO LIMITE DE POSICIONAMENTO AUTOMÁTICO DO SLIDE +CRZ09 OP130;1
   E0609 : BOOL ;	//=DCK_2++ZNE05+CRZ10;POSICIONAMENTO AUTOMÁTICO DO SLIDE TIME-OUT +CRZ10 OP130;1
   E0610 : BOOL ;	//=DCK_2++ZNE05+CRZ11;POSICIONAMENTO AUTOMÁTICO DO SLIDE TIME-OUT +CRZ11 OP130;1
   E0611 : BOOL ;	//=DCK_2++ZNE05+CRZ12;POSICIONAMENTO AUTOMÁTICO DO SLIDE TIME-OUT +CRZ12 OP130;1
   E0612 : BOOL ;	//=DCK_2++ZNE05+PRX02;TIME-OUT DE POSICIONAMENTO AUTOMÁTICO DO PORTAL +PRX02 -OP120;1
   E0613 : BOOL ;
   E0614 : BOOL ;
   E0615 : BOOL ;
   E0616 : BOOL ;	//=DCK_2++ZNE05+HCZ01-U_19;FALHA CARRO MOVIDRIVE +CRX03 - OP130;1
   E0617 : BOOL ;	//=DCK_2++ZNE05+HCZ01-U_20;FALHA MOVIDRIVE SLIDE +CRY05 - OP130;1
   E0618 : BOOL ;	//=DCK_2++ZNE05+HCZ01-U_21;FALHA MOVIDRIVE SLIDE +CRY06 - OP130;1
   E0619 : BOOL ;	//=DCK_2++ZNE05+HCZ01-U_22;FALHA MOVIDRIVE SLIDE +CRZ07 - OP130;1
   E0620 : BOOL ;	//=DCK_2++ZNE05+HCZ01-U_23;FALHA MOVIDRIVE SLIDE +CRZ08 - OP130;1
   E0621 : BOOL ;	//=DCK_2++ZNE05+HCZ01-U_24;FALHA CARRO MOVIDRIVE +CRX04 - OP130;1
   E0622 : BOOL ;	//=DCK_2++ZNE05+HCZ01-U_25;FALHA MOVIDRIVE SLIDE +CRY07 - OP130;1
   E0623 : BOOL ;	//=DCK_2++ZNE05+HCZ01-U_26;FALHA MOVIDRIVE SLIDE +CRY08 - OP130;1
   E0624 : BOOL ;	//=DCK_2++ZNE05+HCZ01-U_27;FALHA MOVIDRIVE SLIDE +CRZ09 - OP130;1
   E0625 : BOOL ;	//=DCK_2++ZNE05+HCZ01-U_28;FALHA MOVIDRIVE SLIDE +CRZ10 - OP130;1
   E0626 : BOOL ;	//=DCK_2++ZNE05+HCZ01-U_29;FALHA MOVIDRIVE SLIDE +CRZ11 - OP130;1
   E0627 : BOOL ;	//=DCK_2++ZNE05+HCZ01-U_30;FALHA MOVIDRIVE SLIDE +CRZ12 - OP130;1
   E0628 : BOOL ;
   E0629 : BOOL ;
   E0630 : BOOL ;
   E0631 : BOOL ;
   E0632 : BOOL ;
   E0633 : BOOL ;
   E0634 : BOOL ;
   E0635 : BOOL ;
   E0636 : BOOL ;
   E0637 : BOOL ;
   E0638 : BOOL ;
   E0639 : BOOL ;
   E0640 : BOOL ;	//=DCK_2++ZNE05+HCZ01-QF_04;MAGNÉTICA DE POTÊNCIA. NOVO PAINEL PARA INSERÇÃO DO MODELO DUV;1
   E0641 : BOOL ;	//=DCK_2++ZNE05+HCZ01-QF_05;MAGNÉTICA DE POTÊNCIA. NOVO PAINEL PARA INSERÇÃO DO MODELO DUV;1
   E0642 : BOOL ;	//=DCK_2++ZNE05+HCZ01-QM_32;MOTOR DESLIZANTE MAGN.INVERSOR +PRY01 OP120;1
   E0643 : BOOL ;	//=DCK_2++ZNE05+HCZ01-QM_33;MOTOR DESLIZANTE MAGN.INVERSOR +PRY02 OP120;1
   E0644 : BOOL ;	//=DCK_2++ZNE05+HCZ01-QM_34;MOTOR DESLIZANTE MAGN.INVERSOR +PRZ04 OP120;1
   E0645 : BOOL ;	//=DCK_2++ZNE05+HCZ01-QF_32;MAGNÉTICA DE POTÊNCIA. NOVO AR CONDICIONADO QE;1
   E0646 : BOOL ;	//=DCK_2++ZNE05+HCZ01-QF_33;MAGNÉTICA DE POTÊNCIA. NOVO AR CONDICIONADO QE;1
   E0647 : BOOL ;	//=DCK_2++ZNE05+HCZ01-QF_89;FREIO DO MOTOR DESLIZANTE MAGN. +PRY01 OP120;1
   E0648 : BOOL ;	//=DCK_2++ZNE05+HCZ01-QF_90;FREIO DO MOTOR DESLIZANTE MAGN. +PRY02 OP120;1
   E0649 : BOOL ;	//=DCK_2++ZNE05+HCZ01-QF_91;FREIO MOTOR DESLIZANTE MAGN. +PRZ04 OP120;1
   E0650 : BOOL ;	//=DCK_2++ZNE05+HCZ01-KA_41;SÉRIE FEEDBACK HABILITA MOVIDRIVE +PRY01 OP120;2
   E0651 : BOOL ;	//=DCK_2++ZNE05+HCZ01-KA_42;SÉRIE FEEDBACK HABILITA MOVIDRIVE +PRY02 OP120;2
   E0652 : BOOL ;	//=DCK_2++ZNE05+HCZ01-KA_43;SÉRIE FEEDBACK HABILITA MOVIDRIVE +PRZ04 OP120;2
   E0653 : BOOL ;
   E0654 : BOOL ;
   E0655 : BOOL ;
   E0656 : BOOL ;	//=DCK_2++ZNE05+PRY01-SQ_01;VIAGEM EXTRA PARA A FRENTE NO SLIDE +PRY01 OP120;1
   E0657 : BOOL ;	//=DCK_2++ZNE05+PRY01-SQ_02;REVERSÃO DE VIAGEM EXTRA NO SLIDE +PRY01 OP120;1
   E0658 : BOOL ;	//=DCK_2++ZNE05+PRY02-SQ_01;VIAGEM EXTRA PARA A FRENTE NO SLIDE +PRY02 OP120;1
   E0659 : BOOL ;	//=DCK_2++ZNE05+PRY02-SQ_02;VIAGEM EXTRA PARA TRÁS NO SLIDE +PRY02 OP120;1
   E0660 : BOOL ;	//=DCK_2++ZNE05+PRZ04-SQ_01;ALTA VIAGEM EXTRA NO SLIDE +PRZ04 OP120;1
   E0661 : BOOL ;	//=DCK_2++ZNE05+PRZ04-SQ_02;BAIXA VIAGEM EXTRA NO SLIDE +PRZ04 OP120;1
   E0662 : BOOL ;	//=DCK_2++ZNE05+PRZ04-SQ_03;HASTE DE CHAVE DE FENDA DE VIAGEM EXTRA NO SLIDE +PRZ04 OP120;1
   E0663 : BOOL ;	//=DCK_2++ZNE05+PRZ04-SQ_05;OTTURATORE DI SICUREZZA +PRZ04 INTERVENUTO OP120
   E0664 : BOOL ;
   E0665 : BOOL ;
   E0666 : BOOL ;
   E0667 : BOOL ;
   E0668 : BOOL ;
   E0669 : BOOL ;
   E0670 : BOOL ;
   E0671 : BOOL ;
   E0672 : BOOL ;	//=DCK_2++ZNE05+HCZ01-U__32;ANOMALIA DE COMUNICAÇÃO MOVIDRIVE +PRY01 OP120;1
   E0673 : BOOL ;	//=DCK_2++ZNE05+HCZ01-U__33;ANOMALIA DE COMUNICAÇÃO MOVIDRIVE +PRY02 OP120;1
   E0674 : BOOL ;	//=DCK_2++ZNE05+HCZ01-U__34;ANOMALIA DE COMUNICAÇÃO MOVIDRIVE +PRZ04 OP120;1
   E0675 : BOOL ;	//=DCK_2++ZNE05+HCZ01-U__32;FALHA MOVIDRIVE SLIDE +PRY01 OP120;1
   E0676 : BOOL ;	//=DCK_2++ZNE05+HCZ01-U__33;FALHA MOVIDRIVE SLIDE +PRY02 OP120;1
   E0677 : BOOL ;	//=DCK_2++ZNE05+HCZ01-U__34;FALHA MOVIDRIVE SLIDE +PRZ04 OP120;1
   E0678 : BOOL ;	//=DCK_2++ZNE05+HCZ01-U__32;AVISO MOVIDRIVE SLIDE +PRY01 OP120;1
   E0679 : BOOL ;	//=DCK_2++ZNE05+HCZ01-U__33;AVISO MOVIDRIVE SLIDE +PRY02 OP120;1
   E0680 : BOOL ;	//=DCK_2++ZNE05+HCZ01-U__34;AVISO MOVIDRIVE SLIDE +PRZ04 OP120;1
   E0681 : BOOL ;	//=DCK_2++ZNE05+HCZ01-U__32;MOVIDRIVE SLIDE +PRY01 NÃO REINICIA OP120;58
   E0682 : BOOL ;	//=DCK_2++ZNE05+HCZ01-U__33;MOVIDRIVE SLIDE +PRY02 NÃO REINICIA OP120;58
   E0683 : BOOL ;	//=DCK_2++ZNE05+HCZ01-U__34;MOVIDRIVE SLIDE +PRZ04 NÃO RESET OP120;58
   E0684 : BOOL ;	//=DCK_2++ZNE05+HCZ01-U__32;DESLIZAMENTO INTERBLOQUEADO DO EIXO MOVIDRIVE +PRY01 OP120;58
   E0685 : BOOL ;	//=DCK_2++ZNE05+HCZ01-U__33;DESLIZAMENTO INTERBLOQUEADO DO EIXO MOVIDRIVE +PRY02 OP120;58
   E0686 : BOOL ;	//=DCK_2++ZNE05+HCZ01-U__34;DESLIZAMENTO INTERBLOQUEADO EIXO MOVIDRIVE +PRZ04 OP120;58
   E0687 : BOOL ;
   E0688 : BOOL ;
   E0689 : BOOL ;
   E0690 : BOOL ;
   E0691 : BOOL ;
   E0692 : BOOL ;
   E0693 : BOOL ;
   E0694 : BOOL ;
   E0695 : BOOL ;
   E0696 : BOOL ;	//=DCK_2++ZNE05+PRY01;POSICIONAMENTO AUTOMÁTICO DO SLIDE TIME-OUT +PRY01 OP120;1
   E0697 : BOOL ;	//=DCK_2++ZNE05+PRY02;POSICIONAMENTO AUTOMÁTICO DO SLIDE TIME-OUT +PRY02 OP120;1
   E0698 : BOOL ;	//=DCK_2++ZNE05+PRZ04;TEMPO LIMITE DE POSICIONAMENTO AUTOMÁTICO DO SLIDE +PRZ04 OP120;1
   E0699 : BOOL ;
   E0700 : BOOL ;
   E0701 : BOOL ;
   E0702 : BOOL ;
   E0703 : BOOL ;
   E0704 : BOOL ;	//=DCK_2++ZNE05+HCZ01-DSW03;NODE 223 PROFINET SCALANCE NOVO GABINETE OP120;1
   E0705 : BOOL ;	//=DCK_2++ZNE05+HCZ01-DMC02;NODE 222 PROFINET ET200S NOVO GABINETE OP120;1
   E0706 : BOOL ;	//=DCK_2++ZNE05+HCZ01-U__32;NÓ 224 PROFINET MOVIDRIVE +PRY01 OP120;1
   E0707 : BOOL ;	//=DCK_2++ZNE05+HCZ01-U__33;NÓ 225 PROFINET MOVIDRIVE +PRY02 OP120;1
   E0708 : BOOL ;	//=DCK_2++ZNE05+HCZ01-U__34;NÓ 226 PROFINET MOVIDRIVE +PRZ04 OP120;1
   E0709 : BOOL ;
   E0710 : BOOL ;
   E0711 : BOOL ;
   E0712 : BOOL ;	//=DCK_2++ZNE05+SWK01-SWK01;ALARME SERVO NÃO ESTÁ OK;1
   E0713 : BOOL ;	//=DCK_2++ZNE05+SWK01-SWK01;ALARME DE COMUNICAÇÃO SERVO NÃO ESTÁ OK;1
   E0714 : BOOL ;	//=DCK_2++ZNE05+SWK01-SWK01;ALARME DE TEMPERATURA DO SERVO NÃO ESTÁ OK;1
   E0715 : BOOL ;	//=DCK_2++ZNE05+SWK01-SWK01;ALARME SERVO;1
   E0716 : BOOL ;	//=DCK_2++ZNE05+SWK01-SWK01;ALARME DE CHAVE DE FENDA NÃO ESTÁ OK;1
   E0717 : BOOL ;	//=DCK_2++ZNE05+SWK01-SWK01;ALARME DE COMUNICAÇÃO DA CHAVE DE FENDA NÃO ESTÁ OK;1
   E0718 : BOOL ;	//=DCK_2++ZNE05+SWK01-SWK01;ALARME DE TEMPERATURA DA CHAVE DE FENDA NÃO ESTÁ OK;1
   E0719 : BOOL ;	//=DCK_2++ZNE05+SWK01-SWK01;ALARME DE CHAVE DE FENDA;1
   E0720 : BOOL ;	//=DCK_2++ZNE05+SWK01-SWK02;ALARME SERVO NÃO ESTÁ OK;1
   E0721 : BOOL ;	//=DCK_2++ZNE05+SWK01-SWK02;ALARME DE COMUNICAÇÃO SERVO NÃO ESTÁ OK;1
   E0722 : BOOL ;	//=DCK_2++ZNE05+SWK01-SWK02;ALARME DE TEMPERATURA DO SERVO NÃO ESTÁ OK;1
   E0723 : BOOL ;	//=DCK_2++ZNE05+SWK01-SWK02;ALARME SERVO;1
   E0724 : BOOL ;	//=DCK_2++ZNE05+SWK01-SWK02;ALARME DE CHAVE DE FENDA NÃO ESTÁ OK;1
   E0725 : BOOL ;	//=DCK_2++ZNE05+SWK01-SWK02;ALARME DE COMUNICAÇÃO DA CHAVE DE FENDA NÃO ESTÁ OK;1
   E0726 : BOOL ;	//=DCK_2++ZNE05+SWK01-SWK02;ALARME DE TEMPERATURA DA CHAVE DE FENDA NÃO ESTÁ OK;1
   E0727 : BOOL ;	//=DCK_2++ZNE05+SWK01-SWK02;ALARME DE CHAVE DE FENDA;1
   E0728 : BOOL ;	//=DCK_2++ZNE05+SWK01-SWK03;ALARME SERVO NÃO ESTÁ OK;1
   E0729 : BOOL ;	//=DCK_2++ZNE05+SWK01-SWK03;ALARME DE COMUNICAÇÃO SERVO NÃO ESTÁ OK;1
   E0730 : BOOL ;	//=DCK_2++ZNE05+SWK01-SWK03;ALARME DE TEMPERATURA DO SERVO NÃO ESTÁ OK;1
   E0731 : BOOL ;	//=DCK_2++ZNE05+SWK01-SWK03;ALARME SERVO;1
   E0732 : BOOL ;	//=DCK_2++ZNE05+SWK01-SWK03;ALARME DE CHAVE DE FENDA NÃO ESTÁ OK;1
   E0733 : BOOL ;	//=DCK_2++ZNE05+SWK01-SWK03;ALARME DE COMUNICAÇÃO DA CHAVE DE FENDA NÃO ESTÁ OK;1
   E0734 : BOOL ;	//=DCK_2++ZNE05+SWK01-SWK03;ALARME DE TEMPERATURA DA CHAVE DE FENDA NÃO ESTÁ OK;1
   E0735 : BOOL ;	//=DCK_2++ZNE05+SWK01-SWK03;ALARME DE CHAVE DE FENDA;1
   E0736 : BOOL ;	//=DCK_2++ZNE05+SWK01-SWK04;ALARME SERVO NÃO ESTÁ OK;1
   E0737 : BOOL ;	//=DCK_2++ZNE05+SWK01-SWK04;ALARME DE COMUNICAÇÃO SERVO NÃO ESTÁ OK;1
   E0738 : BOOL ;	//=DCK_2++ZNE05+SWK01-SWK04;ALARME DE TEMPERATURA DO SERVO NÃO ESTÁ OK;1
   E0739 : BOOL ;	//=DCK_2++ZNE05+SWK01-SWK04;ALARME SERVO;1
   E0740 : BOOL ;	//=DCK_2++ZNE05+SWK01-SWK04;ALARME DE CHAVE DE FENDA NÃO ESTÁ OK;1
   E0741 : BOOL ;	//=DCK_2++ZNE05+SWK01-SWK04;ALARME DE COMUNICAÇÃO DA CHAVE DE FENDA NÃO ESTÁ OK;1
   E0742 : BOOL ;	//=DCK_2++ZNE05+SWK01-SWK04;ALARME DE TEMPERATURA DA CHAVE DE FENDA NÃO ESTÁ OK;1
   E0743 : BOOL ;	//=DCK_2++ZNE05+SWK01-SWK04;ALARME DE CHAVE DE FENDA;1
   E0744 : BOOL ;	//=DCK_2++ZNE05+SWK01-SWK05;ALARME SERVO NÃO ESTÁ OK;1
   E0745 : BOOL ;	//=DCK_2++ZNE05+SWK01-SWK05;ALARME DE COMUNICAÇÃO SERVO NÃO ESTÁ OK;1
   E0746 : BOOL ;	//=DCK_2++ZNE05+SWK01-SWK05;ALARME DE TEMPERATURA DO SERVO NÃO ESTÁ OK;1
   E0747 : BOOL ;	//=DCK_2++ZNE05+SWK01-SWK05;ALARME SERVO;1
   E0748 : BOOL ;	//=DCK_2++ZNE05+SWK01-SWK05;ALARME DE CHAVE DE FENDA NÃO ESTÁ OK;1
   E0749 : BOOL ;	//=DCK_2++ZNE05+SWK01-SWK05;ALARME DE COMUNICAÇÃO DA CHAVE DE FENDA NÃO ESTÁ OK;1
   E0750 : BOOL ;	//=DCK_2++ZNE05+SWK01-SWK05;ALARME DE TEMPERATURA DA CHAVE DE FENDA NÃO ESTÁ OK;1
   E0751 : BOOL ;	//=DCK_2++ZNE05+SWK01-SWK05;ALARME DE CHAVE DE FENDA;1
   E0752 : BOOL ;	//=DCK_2++ZNE05+SWK02-SWK06;ALARME SERVO NÃO ESTÁ OK;1
   E0753 : BOOL ;	//=DCK_2++ZNE05+SWK02-SWK06;ALARME DE COMUNICAÇÃO SERVO NÃO ESTÁ OK;1
   E0754 : BOOL ;	//=DCK_2++ZNE05+SWK02-SWK06;ALARME DE TEMPERATURA DO SERVO NÃO ESTÁ OK;1
   E0755 : BOOL ;	//=DCK_2++ZNE05+SWK02-SWK06;ALARME SERVO;1
   E0756 : BOOL ;	//=DCK_2++ZNE05+SWK02-SWK06;ALARME DE CHAVE DE FENDA NÃO ESTÁ OK;1
   E0757 : BOOL ;	//=DCK_2++ZNE05+SWK02-SWK06;ALARME DE COMUNICAÇÃO DA CHAVE DE FENDA NÃO ESTÁ OK;1
   E0758 : BOOL ;	//=DCK_2++ZNE05+SWK02-SWK06;ALARME DE TEMPERATURA DA CHAVE DE FENDA NÃO ESTÁ OK;1
   E0759 : BOOL ;	//=DCK_2++ZNE05+SWK02-SWK06;ALARME DE CHAVE DE FENDA;1
   E0760 : BOOL ;	//=DCK_2++ZNE05+SWK02-SWK07;ALARME SERVO NÃO ESTÁ OK;1
   E0761 : BOOL ;	//=DCK_2++ZNE05+SWK02-SWK07;ALARME DE COMUNICAÇÃO SERVO NÃO ESTÁ OK;1
   E0762 : BOOL ;	//=DCK_2++ZNE05+SWK02-SWK07;ALARME DE TEMPERATURA DO SERVO NÃO ESTÁ OK;1
   E0763 : BOOL ;	//=DCK_2++ZNE05+SWK02-SWK07;ALARME SERVO;1
   E0764 : BOOL ;	//=DCK_2++ZNE05+SWK02-SWK07;ALARME DE CHAVE DE FENDA NÃO ESTÁ OK;1
   E0765 : BOOL ;	//=DCK_2++ZNE05+SWK02-SWK07;ALARME DE COMUNICAÇÃO DA CHAVE DE FENDA NÃO ESTÁ OK;1
   E0766 : BOOL ;	//=DCK_2++ZNE05+SWK02-SWK07;ALARME DE TEMPERATURA DA CHAVE DE FENDA NÃO ESTÁ OK;1
   E0767 : BOOL ;	//=DCK_2++ZNE05+SWK02-SWK07;ALARME DE CHAVE DE FENDA;1
   E0768 : BOOL ;	//=DCK_2++ZNE05+SWK02-SWK08;ALARME SERVO NÃO ESTÁ OK;1
   E0769 : BOOL ;	//=DCK_2++ZNE05+SWK02-SWK08;ALARME DE COMUNICAÇÃO SERVO NÃO ESTÁ OK;1
   E0770 : BOOL ;	//=DCK_2++ZNE05+SWK02-SWK08;ALARME DE TEMPERATURA DO SERVO NÃO ESTÁ OK;1
   E0771 : BOOL ;	//=DCK_2++ZNE05+SWK02-SWK08;ALARME SERVO;1
   E0772 : BOOL ;	//=DCK_2++ZNE05+SWK02-SWK08;ALARME DE CHAVE DE FENDA NÃO ESTÁ OK;1
   E0773 : BOOL ;	//=DCK_2++ZNE05+SWK02-SWK08;ALARME DE COMUNICAÇÃO DA CHAVE DE FENDA NÃO ESTÁ OK;1
   E0774 : BOOL ;	//=DCK_2++ZNE05+SWK02-SWK08;ALARME DE TEMPERATURA DA CHAVE DE FENDA NÃO ESTÁ OK;1
   E0775 : BOOL ;	//=DCK_2++ZNE05+SWK02-SWK08;ALARME DE CHAVE DE FENDA;1
   E0776 : BOOL ;	//=DCK_2++ZNE05+SWK02-SWK09;ALARME SERVO NÃO ESTÁ OK;1
   E0777 : BOOL ;	//=DCK_2++ZNE05+SWK02-SWK09;ALARME DE COMUNICAÇÃO SERVO NÃO ESTÁ OK;1
   E0778 : BOOL ;	//=DCK_2++ZNE05+SWK02-SWK09;ALARME DE TEMPERATURA DO SERVO NÃO ESTÁ OK;1
   E0779 : BOOL ;	//=DCK_2++ZNE05+SWK02-SWK09;ALARME SERVO;1
   E0780 : BOOL ;	//=DCK_2++ZNE05+SWK02-SWK09;ALARME DE CHAVE DE FENDA NÃO ESTÁ OK;1
   E0781 : BOOL ;	//=DCK_2++ZNE05+SWK02-SWK09;ALARME DE COMUNICAÇÃO DA CHAVE DE FENDA NÃO ESTÁ OK;1
   E0782 : BOOL ;	//=DCK_2++ZNE05+SWK02-SWK09;ALARME DE TEMPERATURA DA CHAVE DE FENDA NÃO ESTÁ OK;1
   E0783 : BOOL ;	//=DCK_2++ZNE05+SWK02-SWK09;ALARME DE CHAVE DE FENDA;1
   E0784 : BOOL ;	//=DCK_2++ZNE05+SWK02-SWK10;ALARME SERVO NÃO ESTÁ OK;1
   E0785 : BOOL ;	//=DCK_2++ZNE05+SWK02-SWK10;ALARME DE COMUNICAÇÃO SERVO NÃO ESTÁ OK;1
   E0786 : BOOL ;	//=DCK_2++ZNE05+SWK02-SWK10;ALARME DE TEMPERATURA DO SERVO NÃO ESTÁ OK;1
   E0787 : BOOL ;	//=DCK_2++ZNE05+SWK02-SWK10;ALARME SERVO;1
   E0788 : BOOL ;	//=DCK_2++ZNE05+SWK02-SWK10;ALARME DE CHAVE DE FENDA NÃO ESTÁ OK;1
   E0789 : BOOL ;	//=DCK_2++ZNE05+SWK02-SWK10;ALARME DE COMUNICAÇÃO DA CHAVE DE FENDA NÃO ESTÁ OK;1
   E0790 : BOOL ;	//=DCK_2++ZNE05+SWK02-SWK10;ALARME DE TEMPERATURA DA CHAVE DE FENDA NÃO ESTÁ OK;1
   E0791 : BOOL ;	//=DCK_2++ZNE05+SWK02-SWK10;ALARME DE CHAVE DE FENDA;1
   E0792 : BOOL ;
   E0793 : BOOL ;
   E0794 : BOOL ;
   E0795 : BOOL ;
   E0796 : BOOL ;
   E0797 : BOOL ;
   E0798 : BOOL ;
   E0799 : BOOL ;
   E0800 : BOOL ;
   E0801 : BOOL ;
   E0802 : BOOL ;
   E0803 : BOOL ;
   E0804 : BOOL ;
   E0805 : BOOL ;
   E0806 : BOOL ;
   E0807 : BOOL ;
   E0808 : BOOL ;
   E0809 : BOOL ;
   E0810 : BOOL ;
   E0811 : BOOL ;
   E0812 : BOOL ;
   E0813 : BOOL ;
   E0814 : BOOL ;
   E0815 : BOOL ;
   E0816 : BOOL ;	//=DCK_2++ZNE05+HCZ01;ALTA TEMPERATURA DO GABINETE;58
   E0817 : BOOL ;
   E0818 : BOOL ;
   E0819 : BOOL ;
   E0820 : BOOL ;
   E0821 : BOOL ;
   E0822 : BOOL ;
   E0823 : BOOL ;
   E0824 : BOOL ;	//=DCK_2++ZNE05+SWK03-SWK01;ALARME SERVO NÃO ESTÁ OK;1
   E0825 : BOOL ;	//=DCK_2++ZNE05+SWK03-SWK01;ALARME DE COMUNICAÇÃO SERVO NÃO ESTÁ OK;1
   E0826 : BOOL ;	//=DCK_2++ZNE05+SWK03-SWK01;ALARME DE TEMPERATURA DO SERVO NÃO ESTÁ OK;1
   E0827 : BOOL ;	//=DCK_2++ZNE05+SWK03-SWK01;ALARME SERVO;1
   E0828 : BOOL ;	//=DCK_2++ZNE05+SWK03-SWK01;ALARME DE CHAVE DE FENDA NÃO ESTÁ OK;1
   E0829 : BOOL ;	//=DCK_2++ZNE05+SWK03-SWK01;ALARME DE COMUNICAÇÃO DA CHAVE DE FENDA NÃO ESTÁ OK;1
   E0830 : BOOL ;	//=DCK_2++ZNE05+SWK03-SWK01;ALARME DE TEMPERATURA DA CHAVE DE FENDA NÃO ESTÁ OK;1
   E0831 : BOOL ;	//=DCK_2++ZNE05+SWK03-SWK01;ALARME DE CHAVE DE FENDA;1
   E0832 : BOOL ;	//=DCK_2++ZNE05+SWK03-SWK02;ALARME SERVO NÃO ESTÁ OK;1
   E0833 : BOOL ;	//=DCK_2++ZNE05+SWK03-SWK02;ALARME DE COMUNICAÇÃO SERVO NÃO ESTÁ OK;1
   E0834 : BOOL ;	//=DCK_2++ZNE05+SWK03-SWK02;ALARME DE TEMPERATURA DO SERVO NÃO ESTÁ OK;1
   E0835 : BOOL ;	//=DCK_2++ZNE05+SWK03-SWK02;ALARME SERVO;1
   E0836 : BOOL ;	//=DCK_2++ZNE05+SWK03-SWK02;ALARME DE CHAVE DE FENDA NÃO ESTÁ OK;1
   E0837 : BOOL ;	//=DCK_2++ZNE05+SWK03-SWK02;ALARME DE COMUNICAÇÃO DA CHAVE DE FENDA NÃO ESTÁ OK;1
   E0838 : BOOL ;	//=DCK_2++ZNE05+SWK03-SWK02;ALARME DE TEMPERATURA DA CHAVE DE FENDA NÃO ESTÁ OK;1
   E0839 : BOOL ;	//=DCK_2++ZNE05+SWK03-SWK02;ALARME DE CHAVE DE FENDA;1
   E0840 : BOOL ;	//=DCK_2++ZNE05+SWK04-SWK03;ALARME SERVO NÃO ESTÁ OK;1
   E0841 : BOOL ;	//=DCK_2++ZNE05+SWK04-SWK03;ALARME DE COMUNICAÇÃO SERVO NÃO ESTÁ OK;1
   E0842 : BOOL ;	//=DCK_2++ZNE05+SWK04-SWK03;ALARME DE TEMPERATURA DO SERVO NÃO ESTÁ OK;1
   E0843 : BOOL ;	//=DCK_2++ZNE05+SWK04-SWK03;ALARME SERVO;1
   E0844 : BOOL ;	//=DCK_2++ZNE05+SWK04-SWK03;ALARME DE CHAVE DE FENDA NÃO ESTÁ OK;1
   E0845 : BOOL ;	//=DCK_2++ZNE05+SWK04-SWK03;ALARME DE COMUNICAÇÃO DA CHAVE DE FENDA NÃO ESTÁ OK;1
   E0846 : BOOL ;	//=DCK_2++ZNE05+SWK04-SWK03;ALARME DE TEMPERATURA DA CHAVE DE FENDA NÃO ESTÁ OK;1
   E0847 : BOOL ;	//=DCK_2++ZNE05+SWK04-SWK03;ALARME DE CHAVE DE FENDA;1
   E0848 : BOOL ;	//=DCK_2++ZNE05+SWK04-SWK04;ALARME SERVO NÃO ESTÁ OK;1
   E0849 : BOOL ;	//=DCK_2++ZNE05+SWK04-SWK04;ALARME DE COMUNICAÇÃO SERVO NÃO ESTÁ OK;1
   E0850 : BOOL ;	//=DCK_2++ZNE05+SWK04-SWK04;ALARME DE TEMPERATURA DO SERVO NÃO ESTÁ OK;1
   E0851 : BOOL ;	//=DCK_2++ZNE05+SWK04-SWK04;ALARME SERVO;1
   E0852 : BOOL ;	//=DCK_2++ZNE05+SWK04-SWK04;ALARME DE CHAVE DE FENDA NÃO ESTÁ OK;1
   E0853 : BOOL ;	//=DCK_2++ZNE05+SWK04-SWK04;ALARME DE COMUNICAÇÃO DA CHAVE DE FENDA NÃO ESTÁ OK;1
   E0854 : BOOL ;	//=DCK_2++ZNE05+SWK04-SWK04;ALARME DE TEMPERATURA DA CHAVE DE FENDA NÃO ESTÁ OK;1
   E0855 : BOOL ;	//=DCK_2++ZNE05+SWK04-SWK04;ALARME DE CHAVE DE FENDA;1
   E0856 : BOOL ;	//=DCK_2++ZNE05+SWK05-SWK05;ALARME SERVO NÃO ESTÁ OK;1
   E0857 : BOOL ;	//=DCK_2++ZNE05+SWK05-SWK05;ALARME DE COMUNICAÇÃO SERVO NÃO ESTÁ OK;1
   E0858 : BOOL ;	//=DCK_2++ZNE05+SWK05-SWK05;ALARME DE TEMPERATURA DO SERVO NÃO ESTÁ OK;1
   E0859 : BOOL ;	//=DCK_2++ZNE05+SWK05-SWK05;ALARME SERVO;1
   E0860 : BOOL ;	//=DCK_2++ZNE05+SWK05-SWK05;ALARME DE CHAVE DE FENDA NÃO ESTÁ OK;1
   E0861 : BOOL ;	//=DCK_2++ZNE05+SWK05-SWK05;ALARME DE COMUNICAÇÃO DA CHAVE DE FENDA NÃO ESTÁ OK;1
   E0862 : BOOL ;	//=DCK_2++ZNE05+SWK05-SWK05;ALARME DE TEMPERATURA DA CHAVE DE FENDA NÃO ESTÁ OK;1
   E0863 : BOOL ;	//=DCK_2++ZNE05+SWK05-SWK05;ALARME DE CHAVE DE FENDA;1
   E0864 : BOOL ;	//=DCK_2++ZNE05+SWK05-SWK06;ALARME SERVO NÃO ESTÁ OK;1
   E0865 : BOOL ;	//=DCK_2++ZNE05+SWK05-SWK06;ALARME DE COMUNICAÇÃO SERVO NÃO ESTÁ OK;1
   E0866 : BOOL ;	//=DCK_2++ZNE05+SWK05-SWK06;ALARME DE TEMPERATURA DO SERVO NÃO ESTÁ OK;1
   E0867 : BOOL ;	//=DCK_2++ZNE05+SWK05-SWK06;ALARME SERVO;1
   E0868 : BOOL ;	//=DCK_2++ZNE05+SWK05-SWK06;ALARME DE CHAVE DE FENDA NÃO ESTÁ OK;1
   E0869 : BOOL ;	//=DCK_2++ZNE05+SWK05-SWK06;ALARME DE COMUNICAÇÃO DA CHAVE DE FENDA NÃO ESTÁ OK;1
   E0870 : BOOL ;	//=DCK_2++ZNE05+SWK05-SWK06;ALARME DE TEMPERATURA DA CHAVE DE FENDA NÃO ESTÁ OK;1
   E0871 : BOOL ;	//=DCK_2++ZNE05+SWK05-SWK06;ALARME DE CHAVE DE FENDA;1
   E0872 : BOOL ;	//=DCK_2++ZNE05+SWK05-SWK07;ALARME SERVO NÃO ESTÁ OK;1
   E0873 : BOOL ;	//=DCK_2++ZNE05+SWK05-SWK07;ALARME DE COMUNICAÇÃO SERVO NÃO ESTÁ OK;1
   E0874 : BOOL ;	//=DCK_2++ZNE05+SWK05-SWK07;ALARME DE TEMPERATURA DO SERVO NÃO ESTÁ OK;1
   E0875 : BOOL ;	//=DCK_2++ZNE05+SWK05-SWK07;ALARME SERVO;1
   E0876 : BOOL ;	//=DCK_2++ZNE05+SWK05-SWK07;ALARME DE CHAVE DE FENDA NÃO ESTÁ OK;1
   E0877 : BOOL ;	//=DCK_2++ZNE05+SWK05-SWK07;ALARME DE COMUNICAÇÃO DA CHAVE DE FENDA NÃO ESTÁ OK;1
   E0878 : BOOL ;	//=DCK_2++ZNE05+SWK05-SWK07;ALARME DE TEMPERATURA DA CHAVE DE FENDA NÃO ESTÁ OK;1
   E0879 : BOOL ;	//=DCK_2++ZNE05+SWK05-SWK07;ALARME DE CHAVE DE FENDA;1
   E0880 : BOOL ;	//=DCK_2++ZNE05+SWK05-SWK08;ALARME SERVO NÃO ESTÁ OK;1
   E0881 : BOOL ;	//=DCK_2++ZNE05+SWK05-SWK08;ALARME DE COMUNICAÇÃO SERVO NÃO ESTÁ OK;1
   E0882 : BOOL ;	//=DCK_2++ZNE05+SWK05-SWK08;ALARME DE TEMPERATURA DO SERVO NÃO ESTÁ OK;1
   E0883 : BOOL ;	//=DCK_2++ZNE05+SWK05-SWK08;ALARME SERVO;1
   E0884 : BOOL ;	//=DCK_2++ZNE05+SWK05-SWK08;ALARME DE CHAVE DE FENDA NÃO ESTÁ OK;1
   E0885 : BOOL ;	//=DCK_2++ZNE05+SWK05-SWK08;ALARME DE COMUNICAÇÃO DA CHAVE DE FENDA NÃO ESTÁ OK;1
   E0886 : BOOL ;	//=DCK_2++ZNE05+SWK05-SWK08;ALARME DE TEMPERATURA DA CHAVE DE FENDA NÃO ESTÁ OK;1
   E0887 : BOOL ;	//=DCK_2++ZNE05+SWK05-SWK08;ALARME DE CHAVE DE FENDA;1
   E0888 : BOOL ;	//=DCK_2++ZNE05+SWK06-SWK09;ALARME SERVO NÃO ESTÁ OK;1
   E0889 : BOOL ;	//=DCK_2++ZNE05+SWK06-SWK09;ALARME DE COMUNICAÇÃO SERVO NÃO ESTÁ OK;1
   E0890 : BOOL ;	//=DCK_2++ZNE05+SWK06-SWK09;ALARME DE TEMPERATURA DO SERVO NÃO ESTÁ OK;1
   E0891 : BOOL ;	//=DCK_2++ZNE05+SWK06-SWK09;ALARME SERVO;1
   E0892 : BOOL ;	//=DCK_2++ZNE05+SWK06-SWK09;ALARME DE CHAVE DE FENDA NÃO ESTÁ OK;1
   E0893 : BOOL ;	//=DCK_2++ZNE05+SWK06-SWK09;ALARME DE COMUNICAÇÃO DA CHAVE DE FENDA NÃO ESTÁ OK;1
   E0894 : BOOL ;	//=DCK_2++ZNE05+SWK06-SWK09;ALARME DE TEMPERATURA DA CHAVE DE FENDA NÃO ESTÁ OK;1
   E0895 : BOOL ;	//=DCK_2++ZNE05+SWK06-SWK09;ALARME DE CHAVE DE FENDA;1
   E0896 : BOOL ;	//=DCK_2++ZNE05+SWK06-SWK10;ALARME SERVO NÃO ESTÁ OK;1
   E0897 : BOOL ;	//=DCK_2++ZNE05+SWK06-SWK10;ALARME DE COMUNICAÇÃO SERVO NÃO ESTÁ OK;1
   E0898 : BOOL ;	//=DCK_2++ZNE05+SWK06-SWK10;ALARME DE TEMPERATURA DO SERVO NÃO ESTÁ OK;1
   E0899 : BOOL ;	//=DCK_2++ZNE05+SWK06-SWK10;ALARME SERVO;1
   E0900 : BOOL ;	//=DCK_2++ZNE05+SWK06-SWK10;ALARME DE CHAVE DE FENDA NÃO ESTÁ OK;1
   E0901 : BOOL ;	//=DCK_2++ZNE05+SWK06-SWK10;ALARME DE COMUNICAÇÃO DA CHAVE DE FENDA NÃO ESTÁ OK;1
   E0902 : BOOL ;	//=DCK_2++ZNE05+SWK06-SWK10;ALARME DE TEMPERATURA DA CHAVE DE FENDA NÃO ESTÁ OK;1
   E0903 : BOOL ;	//=DCK_2++ZNE05+SWK06-SWK10;ALARME DE CHAVE DE FENDA;1
   E0904 : BOOL ;
   E0905 : BOOL ;
   E0906 : BOOL ;
   E0907 : BOOL ;
   E0908 : BOOL ;
   E0909 : BOOL ;
   E0910 : BOOL ;
   E0911 : BOOL ;
   E0912 : BOOL ;	//=DCK_2++ZNE05+CRX01;TRANSPORTE CRX01 EXCLUÍDO SEM BACKUP AUTOMÁTICO;55
   E0913 : BOOL ;	//=DCK_2++ZNE05+CRX02;TRANSPORTE CRX02 EXCLUÍDO SEM BACKUP AUTOMÁTICO;55
   E0914 : BOOL ;	//=DCK_2++ZNE05+CRX03;TRANSPORTE CRX03 EXCLUÍDO SEM BACKUP AUTOMÁTICO;55
   E0915 : BOOL ;	//=DCK_2++ZNE05+CRX04;TRANSPORTE CRX04 EXCLUÍDO SEM BACKUP AUTOMÁTICO;55
   E0916 : BOOL ;
   E0917 : BOOL ;
   E0918 : BOOL ;
   E0919 : BOOL ;
   E0920 : BOOL ;
   E0921 : BOOL ;
   E0922 : BOOL ;
   E0923 : BOOL ;
   E0924 : BOOL ;
   E0925 : BOOL ;
   E0926 : BOOL ;
   E0927 : BOOL ;
   E0928 : BOOL ;
   E0929 : BOOL ;
   E0930 : BOOL ;
   E0931 : BOOL ;
   E0932 : BOOL ;
   E0933 : BOOL ;
   E0934 : BOOL ;
   E0935 : BOOL ;
   E0936 : BOOL ;
   E0937 : BOOL ;
   E0938 : BOOL ;
   E0939 : BOOL ;
   E0940 : BOOL ;
   E0941 : BOOL ;
   E0942 : BOOL ;
   E0943 : BOOL ;
   E0944 : BOOL ;
   E0945 : BOOL ;
   E0946 : BOOL ;
   E0947 : BOOL ;
   E0948 : BOOL ;
   E0949 : BOOL ;
   E0950 : BOOL ;
   E0951 : BOOL ;
   E0952 : BOOL ;
   E0953 : BOOL ;
   E0954 : BOOL ;
   E0955 : BOOL ;
   E0956 : BOOL ;
   E0957 : BOOL ;
   E0958 : BOOL ;
   E0959 : BOOL ;
   E0960 : BOOL ;
   E0961 : BOOL ;
   E0962 : BOOL ;
   E0963 : BOOL ;
   E0964 : BOOL ;
   E0965 : BOOL ;
   E0966 : BOOL ;
   E0967 : BOOL ;
   E0968 : BOOL ;
   E0969 : BOOL ;
   E0970 : BOOL ;
   E0971 : BOOL ;
   E0972 : BOOL ;
   E0973 : BOOL ;
   E0974 : BOOL ;
   E0975 : BOOL ;
   E0976 : BOOL ;
   E0977 : BOOL ;
   E0978 : BOOL ;
   E0979 : BOOL ;
   E0980 : BOOL ;
   E0981 : BOOL ;
   E0982 : BOOL ;
   E0983 : BOOL ;
   E0984 : BOOL ;
   E0985 : BOOL ;
   E0986 : BOOL ;
   E0987 : BOOL ;
   E0988 : BOOL ;
   E0989 : BOOL ;
   E0990 : BOOL ;
   E0991 : BOOL ;
   E0992 : BOOL ;
   E0993 : BOOL ;
   E0994 : BOOL ;
   E0995 : BOOL ;
   E0996 : BOOL ;
   E0997 : BOOL ;
   E0998 : BOOL ;
   E0999 : BOOL ;
   E1000 : BOOL ;
   E1001 : BOOL ;
   E1002 : BOOL ;	//
   E1003 : BOOL ;
   E1004 : BOOL ;
   E1005 : BOOL ;
   E1006 : BOOL ;
   E1007 : BOOL ;
   E1008 : BOOL ;
   E1009 : BOOL ;
   E1010 : BOOL ;
   E1011 : BOOL ;
   E1012 : BOOL ;
   E1013 : BOOL ;
   E1014 : BOOL ;
   E1015 : BOOL ;
   E1016 : BOOL ;
   E1017 : BOOL ;
   E1018 : BOOL ;
   E1019 : BOOL ;
   E1020 : BOOL ;
   E1021 : BOOL ;
   E1022 : BOOL ;
   E1023 : BOOL ;
  END_STRUCT ;
BEGIN
   CM_ID := '=DCK';
   STATION_ID := '++ZNE05';
   ELEMENT_ID := '';
   DB_ID := 3;
   PART_STYLE := '';
   ACT_CYCLE_TIME := 0;
   COUNT_GOOD := 0;
   COUNT_SCRAP := 0;
   SPARE_00[0] := 0;
   SPARE_00[1] := 0;
   SPARE_00[2] := 0;
   SPARE_00[3] := 0;
   SPARE_00[4] := 0;
   SPARE_00[5] := 0;
   SPARE_00[6] := 0;
   SPARE_00[7] := 0;
   SPARE_00[8] := 0;
   SPARE_00[9] := 0;
   SPARE_00[10] := 0;
   SPARE_00[11] := 0;
   SPARE_00[12] := 0;
   SPARE_00[13] := 0;
   SPARE_00[14] := 0;
   SPARE_00[15] := 0;
   SPARE_01[0] := 0;
   SPARE_01[1] := 0;
   SPARE_01[2] := 0;
   SPARE_01[3] := 0;
   SPARE_01[4] := 0;
   SPARE_01[5] := 0;
   SPARE_01[6] := 0;
   SPARE_01[7] := 0;
   SPARE_01[8] := 0;
   SPARE_01[9] := 0;
   SPARE_01[10] := 0;
   SPARE_01[11] := 0;
   SPARE_01[12] := 0;
   SPARE_01[13] := 0;
   SPARE_01[14] := 0;
   SPARE_01[15] := 0;
   SPARE_01[16] := 0;
   SPARE_01[17] := 0;
   CODE_EVENT[0] := 0;
   CODE_EVENT[1] := 0;
   CODE_EVENT[2] := 0;
   CODE_EVENT[3] := 0;
   CODE_EVENT[4] := 0;
   CODE_EVENT[5] := 0;
   CODE_EVENT[6] := 0;
   CODE_EVENT[7] := 0;
   E0000 := FALSE;
   E0001 := FALSE;
   E0002 := FALSE;
   E0003 := FALSE;
   E0004 := FALSE;
   E0005 := FALSE;
   E0006 := FALSE;
   E0007 := FALSE;
   E0008 := FALSE;
   E0009 := FALSE;
   E0010 := FALSE;
   E0011 := FALSE;
   E0012 := FALSE;
   E0013 := FALSE;
   E0014 := FALSE;
   E0015 := FALSE;
   E0016 := FALSE;
   E0017 := FALSE;
   E0018 := FALSE;
   E0019 := FALSE;
   E0020 := FALSE;
   E0021 := FALSE;
   E0022 := FALSE;
   E0023 := FALSE;
   E0024 := FALSE;
   E0025 := FALSE;
   E0026 := FALSE;
   E0027 := FALSE;
   E0028 := FALSE;
   E0029 := FALSE;
   E0030 := FALSE;
   E0031 := FALSE;
   E0032 := FALSE;
   E0033 := FALSE;
   E0034 := FALSE;
   E0035 := FALSE;
   E0036 := FALSE;
   E0037 := FALSE;
   E0038 := FALSE;
   E0039 := FALSE;
   E0040 := FALSE;
   E0041 := FALSE;
   E0042 := FALSE;
   E0043 := FALSE;
   E0044 := FALSE;
   E0045 := FALSE;
   E0046 := FALSE;
   E0047 := FALSE;
   E0048 := FALSE;
   E0049 := FALSE;
   E0050 := FALSE;
   E0051 := FALSE;
   E0052 := FALSE;
   E0053 := FALSE;
   E0054 := FALSE;
   E0055 := FALSE;
   E0056 := FALSE;
   E0057 := FALSE;
   E0058 := FALSE;
   E0059 := FALSE;
   E0060 := FALSE;
   E0061 := FALSE;
   E0062 := FALSE;
   E0063 := FALSE;
   E0064 := FALSE;
   E0065 := FALSE;
   E0066 := FALSE;
   E0067 := FALSE;
   E0068 := FALSE;
   E0069 := FALSE;
   E0070 := FALSE;
   E0071 := FALSE;
   E0072 := FALSE;
   E0073 := FALSE;
   E0074 := FALSE;
   E0075 := FALSE;
   E0076 := FALSE;
   E0077 := FALSE;
   E0078 := FALSE;
   E0079 := FALSE;
   E0080 := FALSE;
   E0081 := FALSE;
   E0082 := FALSE;
   E0083 := FALSE;
   E0084 := FALSE;
   E0085 := FALSE;
   E0086 := FALSE;
   E0087 := FALSE;
   E0088 := FALSE;
   E0089 := FALSE;
   E0090 := FALSE;
   E0091 := FALSE;
   E0092 := FALSE;
   E0093 := FALSE;
   E0094 := FALSE;
   E0095 := FALSE;
   E0096 := FALSE;
   E0097 := FALSE;
   E0098 := FALSE;
   E0099 := FALSE;
   E0100 := FALSE;
   E0101 := FALSE;
   E0102 := FALSE;
   E0103 := FALSE;
   E0104 := FALSE;
   E0105 := FALSE;
   E0106 := FALSE;
   E0107 := FALSE;
   E0108 := FALSE;
   E0109 := FALSE;
   E0110 := FALSE;
   E0111 := FALSE;
   E0112 := FALSE;
   E0113 := FALSE;
   E0114 := FALSE;
   E0115 := FALSE;
   E0116 := FALSE;
   E0117 := FALSE;
   E0118 := FALSE;
   E0119 := FALSE;
   E0120 := FALSE;
   E0121 := FALSE;
   E0122 := FALSE;
   E0123 := FALSE;
   E0124 := FALSE;
   E0125 := FALSE;
   E0126 := FALSE;
   E0127 := FALSE;
   E0128 := FALSE;
   E0129 := FALSE;
   E0130 := FALSE;
   E0131 := FALSE;
   E0132 := FALSE;
   E0133 := FALSE;
   E0134 := FALSE;
   E0135 := FALSE;
   E0136 := FALSE;
   E0137 := FALSE;
   E0138 := FALSE;
   E0139 := FALSE;
   E0140 := FALSE;
   E0141 := FALSE;
   E0142 := FALSE;
   E0143 := FALSE;
   E0144 := FALSE;
   E0145 := FALSE;
   E0146 := FALSE;
   E0147 := FALSE;
   E0148 := FALSE;
   E0149 := FALSE;
   E0150 := FALSE;
   E0151 := FALSE;
   E0152 := FALSE;
   E0153 := FALSE;
   E0154 := FALSE;
   E0155 := FALSE;
   E0156 := FALSE;
   E0157 := FALSE;
   E0158 := FALSE;
   E0159 := FALSE;
   E0160 := FALSE;
   E0161 := FALSE;
   E0162 := FALSE;
   E0163 := FALSE;
   E0164 := FALSE;
   E0165 := FALSE;
   E0166 := FALSE;
   E0167 := FALSE;
   E0168 := FALSE;
   E0169 := FALSE;
   E0170 := FALSE;
   E0171 := FALSE;
   E0172 := FALSE;
   E0173 := FALSE;
   E0174 := FALSE;
   E0175 := FALSE;
   E0176 := FALSE;
   E0177 := FALSE;
   E0178 := FALSE;
   E0179 := FALSE;
   E0180 := FALSE;
   E0181 := FALSE;
   E0182 := FALSE;
   E0183 := FALSE;
   E0184 := FALSE;
   E0185 := FALSE;
   E0186 := FALSE;
   E0187 := FALSE;
   E0188 := FALSE;
   E0189 := FALSE;
   E0190 := FALSE;
   E0191 := FALSE;
   E0192 := FALSE;
   E0193 := FALSE;
   E0194 := FALSE;
   E0195 := FALSE;
   E0196 := FALSE;
   E0197 := FALSE;
   E0198 := FALSE;
   E0199 := FALSE;
   E0200 := FALSE;
   E0201 := FALSE;
   E0202 := FALSE;
   E0203 := FALSE;
   E0204 := FALSE;
   E0205 := FALSE;
   E0206 := FALSE;
   E0207 := FALSE;
   E0208 := FALSE;
   E0209 := FALSE;
   E0210 := FALSE;
   E0211 := FALSE;
   E0212 := FALSE;
   E0213 := FALSE;
   E0214 := FALSE;
   E0215 := FALSE;
   E0216 := FALSE;
   E0217 := FALSE;
   E0218 := FALSE;
   E0219 := FALSE;
   E0220 := FALSE;
   E0221 := FALSE;
   E0222 := FALSE;
   E0223 := FALSE;
   E0224 := FALSE;
   E0225 := FALSE;
   E0226 := FALSE;
   E0227 := FALSE;
   E0228 := FALSE;
   E0229 := FALSE;
   E0230 := FALSE;
   E0231 := FALSE;
   E0232 := FALSE;
   E0233 := FALSE;
   E0234 := FALSE;
   E0235 := FALSE;
   E0236 := FALSE;
   E0237 := FALSE;
   E0238 := FALSE;
   E0239 := FALSE;
   E0240 := FALSE;
   E0241 := FALSE;
   E0242 := FALSE;
   E0243 := FALSE;
   E0244 := FALSE;
   E0245 := FALSE;
   E0246 := FALSE;
   E0247 := FALSE;
   E0248 := FALSE;
   E0249 := FALSE;
   E0250 := FALSE;
   E0251 := FALSE;
   E0252 := FALSE;
   E0253 := FALSE;
   E0254 := FALSE;
   E0255 := FALSE;
   E0256 := FALSE;
   E0257 := FALSE;
   E0258 := FALSE;
   E0259 := FALSE;
   E0260 := FALSE;
   E0261 := FALSE;
   E0262 := FALSE;
   E0263 := FALSE;
   E0264 := FALSE;
   E0265 := FALSE;
   E0266 := FALSE;
   E0267 := FALSE;
   E0268 := FALSE;
   E0269 := FALSE;
   E0270 := FALSE;
   E0271 := FALSE;
   E0272 := FALSE;
   E0273 := FALSE;
   E0274 := FALSE;
   E0275 := FALSE;
   E0276 := FALSE;
   E0277 := FALSE;
   E0278 := FALSE;
   E0279 := FALSE;
   E0280 := FALSE;
   E0281 := FALSE;
   E0282 := FALSE;
   E0283 := FALSE;
   E0284 := FALSE;
   E0285 := FALSE;
   E0286 := FALSE;
   E0287 := FALSE;
   E0288 := FALSE;
   E0289 := FALSE;
   E0290 := FALSE;
   E0291 := FALSE;
   E0292 := FALSE;
   E0293 := FALSE;
   E0294 := FALSE;
   E0295 := FALSE;
   E0296 := FALSE;
   E0297 := FALSE;
   E0298 := FALSE;
   E0299 := FALSE;
   E0300 := FALSE;
   E0301 := FALSE;
   E0302 := FALSE;
   E0303 := FALSE;
   E0304 := FALSE;
   E0305 := FALSE;
   E0306 := FALSE;
   E0307 := FALSE;
   E0308 := FALSE;
   E0309 := FALSE;
   E0310 := FALSE;
   E0311 := FALSE;
   E0312 := FALSE;
   E0313 := FALSE;
   E0314 := FALSE;
   E0315 := FALSE;
   E0316 := FALSE;
   E0317 := FALSE;
   E0318 := FALSE;
   E0319 := FALSE;
   E0320 := FALSE;
   E0321 := FALSE;
   E0322 := FALSE;
   E0323 := FALSE;
   E0324 := FALSE;
   E0325 := FALSE;
   E0326 := FALSE;
   E0327 := FALSE;
   E0328 := FALSE;
   E0329 := FALSE;
   E0330 := FALSE;
   E0331 := FALSE;
   E0332 := FALSE;
   E0333 := FALSE;
   E0334 := FALSE;
   E0335 := FALSE;
   E0336 := FALSE;
   E0337 := FALSE;
   E0338 := FALSE;
   E0339 := FALSE;
   E0340 := FALSE;
   E0341 := FALSE;
   E0342 := FALSE;
   E0343 := FALSE;
   E0344 := FALSE;
   E0345 := FALSE;
   E0346 := FALSE;
   E0347 := FALSE;
   E0348 := FALSE;
   E0349 := FALSE;
   E0350 := FALSE;
   E0351 := FALSE;
   E0352 := FALSE;
   E0353 := FALSE;
   E0354 := FALSE;
   E0355 := FALSE;
   E0356 := FALSE;
   E0357 := FALSE;
   E0358 := FALSE;
   E0359 := FALSE;
   E0360 := FALSE;
   E0361 := FALSE;
   E0362 := FALSE;
   E0363 := FALSE;
   E0364 := FALSE;
   E0365 := FALSE;
   E0366 := FALSE;
   E0367 := FALSE;
   E0368 := FALSE;
   E0369 := FALSE;
   E0370 := FALSE;
   E0371 := FALSE;
   E0372 := FALSE;
   E0373 := FALSE;
   E0374 := FALSE;
   E0375 := FALSE;
   E0376 := FALSE;
   E0377 := FALSE;
   E0378 := FALSE;
   E0379 := FALSE;
   E0380 := FALSE;
   E0381 := FALSE;
   E0382 := FALSE;
   E0383 := FALSE;
   E0384 := FALSE;
   E0385 := FALSE;
   E0386 := FALSE;
   E0387 := FALSE;
   E0388 := FALSE;
   E0389 := FALSE;
   E0390 := FALSE;
   E0391 := FALSE;
   E0392 := FALSE;
   E0393 := FALSE;
   E0394 := FALSE;
   E0395 := FALSE;
   E0396 := FALSE;
   E0397 := FALSE;
   E0398 := FALSE;
   E0399 := FALSE;
   E0400 := FALSE;
   E0401 := FALSE;
   E0402 := FALSE;
   E0403 := FALSE;
   E0404 := FALSE;
   E0405 := FALSE;
   E0406 := FALSE;
   E0407 := FALSE;
   E0408 := FALSE;
   E0409 := FALSE;
   E0410 := FALSE;
   E0411 := FALSE;
   E0412 := FALSE;
   E0413 := FALSE;
   E0414 := FALSE;
   E0415 := FALSE;
   E0416 := FALSE;
   E0417 := FALSE;
   E0418 := FALSE;
   E0419 := FALSE;
   E0420 := FALSE;
   E0421 := FALSE;
   E0422 := FALSE;
   E0423 := FALSE;
   E0424 := FALSE;
   E0425 := FALSE;
   E0426 := FALSE;
   E0427 := FALSE;
   E0428 := FALSE;
   E0429 := FALSE;
   E0430 := FALSE;
   E0431 := FALSE;
   E0432 := FALSE;
   E0433 := FALSE;
   E0434 := FALSE;
   E0435 := FALSE;
   E0436 := FALSE;
   E0437 := FALSE;
   E0438 := FALSE;
   E0439 := FALSE;
   E0440 := FALSE;
   E0441 := FALSE;
   E0442 := FALSE;
   E0443 := FALSE;
   E0444 := FALSE;
   E0445 := FALSE;
   E0446 := FALSE;
   E0447 := FALSE;
   E0448 := FALSE;
   E0449 := FALSE;
   E0450 := FALSE;
   E0451 := FALSE;
   E0452 := FALSE;
   E0453 := FALSE;
   E0454 := FALSE;
   E0455 := FALSE;
   E0456 := FALSE;
   E0457 := FALSE;
   E0458 := FALSE;
   E0459 := FALSE;
   E0460 := FALSE;
   E0461 := FALSE;
   E0462 := FALSE;
   E0463 := FALSE;
   E0464 := FALSE;
   E0465 := FALSE;
   E0466 := FALSE;
   E0467 := FALSE;
   E0468 := FALSE;
   E0469 := FALSE;
   E0470 := FALSE;
   E0471 := FALSE;
   E0472 := FALSE;
   E0473 := FALSE;
   E0474 := FALSE;
   E0475 := FALSE;
   E0476 := FALSE;
   E0477 := FALSE;
   E0478 := FALSE;
   E0479 := FALSE;
   E0480 := FALSE;
   E0481 := FALSE;
   E0482 := FALSE;
   E0483 := FALSE;
   E0484 := FALSE;
   E0485 := FALSE;
   E0486 := FALSE;
   E0487 := FALSE;
   E0488 := FALSE;
   E0489 := FALSE;
   E0490 := FALSE;
   E0491 := FALSE;
   E0492 := FALSE;
   E0493 := FALSE;
   E0494 := FALSE;
   E0495 := FALSE;
   E0496 := FALSE;
   E0497 := FALSE;
   E0498 := FALSE;
   E0499 := FALSE;
   E0500 := FALSE;
   E0501 := FALSE;
   E0502 := FALSE;
   E0503 := FALSE;
   E0504 := FALSE;
   E0505 := FALSE;
   E0506 := FALSE;
   E0507 := FALSE;
   E0508 := FALSE;
   E0509 := FALSE;
   E0510 := FALSE;
   E0511 := FALSE;
   E0512 := FALSE;
   E0513 := FALSE;
   E0514 := FALSE;
   E0515 := FALSE;
   E0516 := FALSE;
   E0517 := FALSE;
   E0518 := FALSE;
   E0519 := FALSE;
   E0520 := FALSE;
   E0521 := FALSE;
   E0522 := FALSE;
   E0523 := FALSE;
   E0524 := FALSE;
   E0525 := FALSE;
   E0526 := FALSE;
   E0527 := FALSE;
   E0528 := FALSE;
   E0529 := FALSE;
   E0530 := FALSE;
   E0531 := FALSE;
   E0532 := FALSE;
   E0533 := FALSE;
   E0534 := FALSE;
   E0535 := FALSE;
   E0536 := FALSE;
   E0537 := FALSE;
   E0538 := FALSE;
   E0539 := FALSE;
   E0540 := FALSE;
   E0541 := FALSE;
   E0542 := FALSE;
   E0543 := FALSE;
   E0544 := FALSE;
   E0545 := FALSE;
   E0546 := FALSE;
   E0547 := FALSE;
   E0548 := FALSE;
   E0549 := FALSE;
   E0550 := FALSE;
   E0551 := FALSE;
   E0552 := FALSE;
   E0553 := FALSE;
   E0554 := FALSE;
   E0555 := FALSE;
   E0556 := FALSE;
   E0557 := FALSE;
   E0558 := FALSE;
   E0559 := FALSE;
   E0560 := FALSE;
   E0561 := FALSE;
   E0562 := FALSE;
   E0563 := FALSE;
   E0564 := FALSE;
   E0565 := FALSE;
   E0566 := FALSE;
   E0567 := FALSE;
   E0568 := FALSE;
   E0569 := FALSE;
   E0570 := FALSE;
   E0571 := FALSE;
   E0572 := FALSE;
   E0573 := FALSE;
   E0574 := FALSE;
   E0575 := FALSE;
   E0576 := FALSE;
   E0577 := FALSE;
   E0578 := FALSE;
   E0579 := FALSE;
   E0580 := FALSE;
   E0581 := FALSE;
   E0582 := FALSE;
   E0583 := FALSE;
   E0584 := FALSE;
   E0585 := FALSE;
   E0586 := FALSE;
   E0587 := FALSE;
   E0588 := FALSE;
   E0589 := FALSE;
   E0590 := FALSE;
   E0591 := FALSE;
   E0592 := FALSE;
   E0593 := FALSE;
   E0594 := FALSE;
   E0595 := FALSE;
   E0596 := FALSE;
   E0597 := FALSE;
   E0598 := FALSE;
   E0599 := FALSE;
   E0600 := FALSE;
   E0601 := FALSE;
   E0602 := FALSE;
   E0603 := FALSE;
   E0604 := FALSE;
   E0605 := FALSE;
   E0606 := FALSE;
   E0607 := FALSE;
   E0608 := FALSE;
   E0609 := FALSE;
   E0610 := FALSE;
   E0611 := FALSE;
   E0612 := FALSE;
   E0613 := FALSE;
   E0614 := FALSE;
   E0615 := FALSE;
   E0616 := FALSE;
   E0617 := FALSE;
   E0618 := FALSE;
   E0619 := FALSE;
   E0620 := FALSE;
   E0621 := FALSE;
   E0622 := FALSE;
   E0623 := FALSE;
   E0624 := FALSE;
   E0625 := FALSE;
   E0626 := FALSE;
   E0627 := FALSE;
   E0628 := FALSE;
   E0629 := FALSE;
   E0630 := FALSE;
   E0631 := FALSE;
   E0632 := FALSE;
   E0633 := FALSE;
   E0634 := FALSE;
   E0635 := FALSE;
   E0636 := FALSE;
   E0637 := FALSE;
   E0638 := FALSE;
   E0639 := FALSE;
   E0640 := FALSE;
   E0641 := FALSE;
   E0642 := FALSE;
   E0643 := FALSE;
   E0644 := FALSE;
   E0645 := FALSE;
   E0646 := FALSE;
   E0647 := FALSE;
   E0648 := FALSE;
   E0649 := FALSE;
   E0650 := FALSE;
   E0651 := FALSE;
   E0652 := FALSE;
   E0653 := FALSE;
   E0654 := FALSE;
   E0655 := FALSE;
   E0656 := FALSE;
   E0657 := FALSE;
   E0658 := FALSE;
   E0659 := FALSE;
   E0660 := FALSE;
   E0661 := FALSE;
   E0662 := FALSE;
   E0663 := FALSE;
   E0664 := FALSE;
   E0665 := FALSE;
   E0666 := FALSE;
   E0667 := FALSE;
   E0668 := FALSE;
   E0669 := FALSE;
   E0670 := FALSE;
   E0671 := FALSE;
   E0672 := FALSE;
   E0673 := FALSE;
   E0674 := FALSE;
   E0675 := FALSE;
   E0676 := FALSE;
   E0677 := FALSE;
   E0678 := FALSE;
   E0679 := FALSE;
   E0680 := FALSE;
   E0681 := FALSE;
   E0682 := FALSE;
   E0683 := FALSE;
   E0684 := FALSE;
   E0685 := FALSE;
   E0686 := FALSE;
   E0687 := FALSE;
   E0688 := FALSE;
   E0689 := FALSE;
   E0690 := FALSE;
   E0691 := FALSE;
   E0692 := FALSE;
   E0693 := FALSE;
   E0694 := FALSE;
   E0695 := FALSE;
   E0696 := FALSE;
   E0697 := FALSE;
   E0698 := FALSE;
   E0699 := FALSE;
   E0700 := FALSE;
   E0701 := FALSE;
   E0702 := FALSE;
   E0703 := FALSE;
   E0704 := FALSE;
   E0705 := FALSE;
   E0706 := FALSE;
   E0707 := FALSE;
   E0708 := FALSE;
   E0709 := FALSE;
   E0710 := FALSE;
   E0711 := FALSE;
   E0712 := FALSE;
   E0713 := FALSE;
   E0714 := FALSE;
   E0715 := FALSE;
   E0716 := FALSE;
   E0717 := FALSE;
   E0718 := FALSE;
   E0719 := FALSE;
   E0720 := FALSE;
   E0721 := FALSE;
   E0722 := FALSE;
   E0723 := FALSE;
   E0724 := FALSE;
   E0725 := FALSE;
   E0726 := FALSE;
   E0727 := FALSE;
   E0728 := FALSE;
   E0729 := FALSE;
   E0730 := FALSE;
   E0731 := FALSE;
   E0732 := FALSE;
   E0733 := FALSE;
   E0734 := FALSE;
   E0735 := FALSE;
   E0736 := FALSE;
   E0737 := FALSE;
   E0738 := FALSE;
   E0739 := FALSE;
   E0740 := FALSE;
   E0741 := FALSE;
   E0742 := FALSE;
   E0743 := FALSE;
   E0744 := FALSE;
   E0745 := FALSE;
   E0746 := FALSE;
   E0747 := FALSE;
   E0748 := FALSE;
   E0749 := FALSE;
   E0750 := FALSE;
   E0751 := FALSE;
   E0752 := FALSE;
   E0753 := FALSE;
   E0754 := FALSE;
   E0755 := FALSE;
   E0756 := FALSE;
   E0757 := FALSE;
   E0758 := FALSE;
   E0759 := FALSE;
   E0760 := FALSE;
   E0761 := FALSE;
   E0762 := FALSE;
   E0763 := FALSE;
   E0764 := FALSE;
   E0765 := FALSE;
   E0766 := FALSE;
   E0767 := FALSE;
   E0768 := FALSE;
   E0769 := FALSE;
   E0770 := FALSE;
   E0771 := FALSE;
   E0772 := FALSE;
   E0773 := FALSE;
   E0774 := FALSE;
   E0775 := FALSE;
   E0776 := FALSE;
   E0777 := FALSE;
   E0778 := FALSE;
   E0779 := FALSE;
   E0780 := FALSE;
   E0781 := FALSE;
   E0782 := FALSE;
   E0783 := FALSE;
   E0784 := FALSE;
   E0785 := FALSE;
   E0786 := FALSE;
   E0787 := FALSE;
   E0788 := FALSE;
   E0789 := FALSE;
   E0790 := FALSE;
   E0791 := FALSE;
   E0792 := FALSE;
   E0793 := FALSE;
   E0794 := FALSE;
   E0795 := FALSE;
   E0796 := FALSE;
   E0797 := FALSE;
   E0798 := FALSE;
   E0799 := FALSE;
   E0800 := FALSE;
   E0801 := FALSE;
   E0802 := FALSE;
   E0803 := FALSE;
   E0804 := FALSE;
   E0805 := FALSE;
   E0806 := FALSE;
   E0807 := FALSE;
   E0808 := FALSE;
   E0809 := FALSE;
   E0810 := FALSE;
   E0811 := FALSE;
   E0812 := FALSE;
   E0813 := FALSE;
   E0814 := FALSE;
   E0815 := FALSE;
   E0816 := FALSE;
   E0817 := FALSE;
   E0818 := FALSE;
   E0819 := FALSE;
   E0820 := FALSE;
   E0821 := FALSE;
   E0822 := FALSE;
   E0823 := FALSE;
   E0824 := FALSE;
   E0825 := FALSE;
   E0826 := FALSE;
   E0827 := FALSE;
   E0828 := FALSE;
   E0829 := FALSE;
   E0830 := FALSE;
   E0831 := FALSE;
   E0832 := FALSE;
   E0833 := FALSE;
   E0834 := FALSE;
   E0835 := FALSE;
   E0836 := FALSE;
   E0837 := FALSE;
   E0838 := FALSE;
   E0839 := FALSE;
   E0840 := FALSE;
   E0841 := FALSE;
   E0842 := FALSE;
   E0843 := FALSE;
   E0844 := FALSE;
   E0845 := FALSE;
   E0846 := FALSE;
   E0847 := FALSE;
   E0848 := FALSE;
   E0849 := FALSE;
   E0850 := FALSE;
   E0851 := FALSE;
   E0852 := FALSE;
   E0853 := FALSE;
   E0854 := FALSE;
   E0855 := FALSE;
   E0856 := FALSE;
   E0857 := FALSE;
   E0858 := FALSE;
   E0859 := FALSE;
   E0860 := FALSE;
   E0861 := FALSE;
   E0862 := FALSE;
   E0863 := FALSE;
   E0864 := FALSE;
   E0865 := FALSE;
   E0866 := FALSE;
   E0867 := FALSE;
   E0868 := FALSE;
   E0869 := FALSE;
   E0870 := FALSE;
   E0871 := FALSE;
   E0872 := FALSE;
   E0873 := FALSE;
   E0874 := FALSE;
   E0875 := FALSE;
   E0876 := FALSE;
   E0877 := FALSE;
   E0878 := FALSE;
   E0879 := FALSE;
   E0880 := FALSE;
   E0881 := FALSE;
   E0882 := FALSE;
   E0883 := FALSE;
   E0884 := FALSE;
   E0885 := FALSE;
   E0886 := FALSE;
   E0887 := FALSE;
   E0888 := FALSE;
   E0889 := FALSE;
   E0890 := FALSE;
   E0891 := FALSE;
   E0892 := FALSE;
   E0893 := FALSE;
   E0894 := FALSE;
   E0895 := FALSE;
   E0896 := FALSE;
   E0897 := FALSE;
   E0898 := FALSE;
   E0899 := FALSE;
   E0900 := FALSE;
   E0901 := FALSE;
   E0902 := FALSE;
   E0903 := FALSE;
   E0904 := FALSE;
   E0905 := FALSE;
   E0906 := FALSE;
   E0907 := FALSE;
   E0908 := FALSE;
   E0909 := FALSE;
   E0910 := FALSE;
   E0911 := FALSE;
   E0912 := FALSE;
   E0913 := FALSE;
   E0914 := FALSE;
   E0915 := FALSE;
   E0916 := FALSE;
   E0917 := FALSE;
   E0918 := FALSE;
   E0919 := FALSE;
   E0920 := FALSE;
   E0921 := FALSE;
   E0922 := FALSE;
   E0923 := FALSE;
   E0924 := FALSE;
   E0925 := FALSE;
   E0926 := FALSE;
   E0927 := FALSE;
   E0928 := FALSE;
   E0929 := FALSE;
   E0930 := FALSE;
   E0931 := FALSE;
   E0932 := FALSE;
   E0933 := FALSE;
   E0934 := FALSE;
   E0935 := FALSE;
   E0936 := FALSE;
   E0937 := FALSE;
   E0938 := FALSE;
   E0939 := FALSE;
   E0940 := FALSE;
   E0941 := FALSE;
   E0942 := FALSE;
   E0943 := FALSE;
   E0944 := FALSE;
   E0945 := FALSE;
   E0946 := FALSE;
   E0947 := FALSE;
   E0948 := FALSE;
   E0949 := FALSE;
   E0950 := FALSE;
   E0951 := FALSE;
   E0952 := FALSE;
   E0953 := FALSE;
   E0954 := FALSE;
   E0955 := FALSE;
   E0956 := FALSE;
   E0957 := FALSE;
   E0958 := FALSE;
   E0959 := FALSE;
   E0960 := FALSE;
   E0961 := FALSE;
   E0962 := FALSE;
   E0963 := FALSE;
   E0964 := FALSE;
   E0965 := FALSE;
   E0966 := FALSE;
   E0967 := FALSE;
   E0968 := FALSE;
   E0969 := FALSE;
   E0970 := FALSE;
   E0971 := FALSE;
   E0972 := FALSE;
   E0973 := FALSE;
   E0974 := FALSE;
   E0975 := FALSE;
   E0976 := FALSE;
   E0977 := FALSE;
   E0978 := FALSE;
   E0979 := FALSE;
   E0980 := FALSE;
   E0981 := FALSE;
   E0982 := FALSE;
   E0983 := FALSE;
   E0984 := FALSE;
   E0985 := FALSE;
   E0986 := FALSE;
   E0987 := FALSE;
   E0988 := FALSE;
   E0989 := FALSE;
   E0990 := FALSE;
   E0991 := FALSE;
   E0992 := FALSE;
   E0993 := FALSE;
   E0994 := FALSE;
   E0995 := FALSE;
   E0996 := FALSE;
   E0997 := FALSE;
   E0998 := FALSE;
   E0999 := FALSE;
   E1000 := FALSE;
   E1001 := FALSE;
   E1002 := FALSE;
   E1003 := FALSE;
   E1004 := FALSE;
   E1005 := FALSE;
   E1006 := FALSE;
   E1007 := FALSE;
   E1008 := FALSE;
   E1009 := FALSE;
   E1010 := FALSE;
   E1011 := FALSE;
   E1012 := FALSE;
   E1013 := FALSE;
   E1014 := FALSE;
   E1015 := FALSE;
   E1016 := FALSE;
   E1017 := FALSE;
   E1018 := FALSE;
   E1019 := FALSE;
   E1020 := FALSE;
   E1021 := FALSE;
   E1022 := FALSE;
   E1023 := FALSE;
END_DATA_BLOCK
